// Safe interface assignments
iTestCommand := TestCommand[TestIdx];

iTestCommandConfig := TestCommandConfig[TestIdx];

iTestComponent := TestComponent[TestIdx];

iTestPermIntlkConfig := TestCommandConfig[TestIdx];

IF iTestCommandConfig <> 0 THEN
	stCommandStatus.ConfigRef REF= iTestCommandConfig.P_CommandConfiguration;
END_IF

IF iTestPermIntlkConfig <> 0 THEN
    iTestPermIntlkConfig.P_PermIntlkConfiguration.PermIntlkObj[1].Description := 'Test Permissive';
    iTestPermIntlkConfig.P_PermIntlkConfiguration.PermIntlkObj[1].Condition := TRUE;
    iTestPermIntlkConfig.P_PermIntlkConfiguration.PermIntlkObj[1].Index := 1;
END_IF

// Configure command
iTestCommandConfig.P_CommandConfiguration.CommandDescription := 'Method Enablement Test - Done State Methods';

// Setup command with configurations
iTestCommand.InjectConfigurations(
    iComponent := iTestComponent,
    iCommandConfiguration := iTestCommandConfig,
    iPermIntlkConfiguration := iTestPermIntlkConfig
);

// Create InputMask 4 state: Done=TRUE, all others FALSE
stCommandStatus.BaseStatus.Busy := FALSE;
stCommandStatus.BaseStatus.Error := FALSE;
stCommandStatus.BaseStatus.Done := TRUE;    // Bit 2 = InputMask 4
stCommandStatus.ConfigRef.PermIntlkConfiguredAsInterlock := FALSE;
stCommandStatus.ConfigRef.AbortOnInterlockDrop := FALSE;
// TRUE := FALSE;
// FALSE := FALSE;

// Inject done state
iTestCommand.SetCommandStatus(stCommandStatus);

// REAL TEST 1: Try Reset() - should succeed in done state
iTestCommand.Reset();

// Verify Reset was accepted
AssertEquals_UDINT(
    Expected := E_CommandResult.None,
    Actual := iTestCommand.P_CommandStatus.Result,
    Message := 'Reset should be accepted in done state (InputMask 4)'
);

// Verify Reset cleared the done state
AssertEquals_UDINT(
    Expected := E_CommandState.Idle,
    Actual := iTestCommand.P_CommandStatus.StepState,
    Message := 'Reset should transition command back to idle state'
);

// Reset to done state for second test
stCommandStatus.BaseStatus.Done := TRUE;
iTestCommand.SetCommandStatus(stCommandStatus);

// REAL TEST 2: Try Execute() - should fail in done state
iTestCommand.Execute();

// Verify Execute was rejected (Result remains unchanged when Done=TRUE)
AssertEquals_UDINT(
    Expected := E_CommandResult.None,
    Actual := iTestCommand.P_CommandStatus.Result,
    Message := 'Execute should be rejected in done state - Result remains unchanged (InputMask 4)'
);

TEST_FINISHED();
END_METHOD

METHOD PRIVATE TEST_MethodEnablement_IdleWithInterlockOK_ShouldAllowExecute
VAR
	TestIdx : DINT := INDEX_METHODENABLEMENT_IDLEWITHINTERLOK_ALLOWEXECUTE;
    stCommandStatus : ST_CommandStatus;
	stBaseStatus	: ST_BaseStatus;
    eResult : E_CommandResult;
END_VAR
TEST(__POUNAME());

// REAL TEST: InputMask 32 (Idle + PermIntlkOK=1) should enable Execute
// From CSV: EnabledMethods="Execute,Cancel,Resume,Queue,Validate"

// Initialize test objects
TestCommand[TestIdx].Initialize();
TestComponent[TestIdx].Initialize();
TestCommandConfig[TestIdx].Initialize();

stCommandStatus.BaseStatus REF= stBaseStatus;

// Safe interface assignments
iTestCommand := TestCommand[TestIdx];

iTestCommandConfig := TestCommandConfig[TestIdx];

iTestComponent := TestComponent[TestIdx];

iTestPermIntlkConfig := TestCommandConfig[TestIdx];

IF iTestCommandConfig <> 0 THEN
	stCommandStatus.ConfigRef REF= iTestCommandConfig.P_CommandConfiguration;
END_IF

IF iTestPermIntlkConfig <> 0 THEN
    iTestPermIntlkConfig.P_PermIntlkConfiguration.PermIntlkObj[1].Description := 'Test Permissive';
    iTestPermIntlkConfig.P_PermIntlkConfiguration.PermIntlkObj[1].Condition := TRUE;
    iTestPermIntlkConfig.P_PermIntlkConfiguration.PermIntlkObj[1].Index := 1;
END_IF

// Configure command with interlock
iTestCommandConfig.P_CommandConfiguration.CommandDescription := 'Method Enablement Test - Execute with Interlock OK';

// Setup command with configurations
iTestCommand.InjectConfigurations(
    iComponent := iTestComponent,
    iCommandConfiguration := iTestCommandConfig,
    iPermIntlkConfiguration := iTestPermIntlkConfig
);

// Create InputMask 32 state: Idle but with PermIntlkOK=1
stCommandStatus.BaseStatus.Busy := FALSE;
stCommandStatus.BaseStatus.Error := FALSE;
stCommandStatus.BaseStatus.Done := FALSE;
stCommandStatus.ConfigRef.PermIntlkConfiguredAsInterlock := FALSE;
stCommandStatus.ConfigRef.AbortOnInterlockDrop := FALSE;
// TRUE := TRUE;  // Bit 5 = InputMask 32
// FALSE := FALSE;

// Inject this specific state
iTestCommand.SetCommandStatus(stCommandStatus);

// First validate the command (component pattern: validate then execute)
iTestCommand.Validate();

// Verify validation succeeded
AssertEquals_UDINT(
    Expected := E_CommandResult.Accepted,
    Actual := iTestCommand.P_CommandStatus.Result,
    Message := 'Command should be Accepted after validation with PermIntlkOK=TRUE'
);

// REAL TEST: Try Execute() - should succeed per truth table
iTestCommand.Execute();

// Verify Execute was accepted (should still be Accepted)
AssertEquals_UDINT(
    Expected := E_CommandResult.Accepted,
    Actual := iTestCommand.P_CommandStatus.Result,
    Message := 'Execute should maintain Accepted state when transitioning from Idle to Execute'
);

// Verify command status reflects execution
AssertTrue(
    Condition := iTestCommand.P_CommandStatus.BaseStatus.Busy OR 
                 iTestCommand.P_CommandStatus.StepState <> E_CommandState.Idle,
    Message := 'Command should transition from idle after successful Execute()'
);

TEST_FINISHED();
END_METHOD

METHOD PRIVATE TEST_MethodEnablement_IdleWithoutInterlockOK_ShouldRejectExecute
VAR
	TestIdx : DINT := INDEX_METHODENABLEMENT_IDLEWITHOUTINTERLOK_REJECT;
    stCommandStatus : ST_CommandStatus;
	stBaseStatus	: ST_BaseStatus;
    stCommandConfiguration : ST_CommandConfiguration;
    eResult : E_CommandResult;
END_VAR
TEST(__POUNAME());

// REAL TEST: InputMask 0 (Idle + PermIntlkOK=0) should reject Execute
// From CSV: EnabledMethods="Cancel,Resume,Queue" (Execute NOT enabled)

// Initialize test objects
TestCommand[TestIdx].Initialize();
TestComponent[TestIdx].Initialize();
TestCommandConfig[TestIdx].Initialize();

stCommandStatus.BaseStatus REF= stBaseStatus;

// Safe interface assignments
iTestCommand := TestCommand[TestIdx];

iTestCommandConfig := TestCommandConfig[TestIdx];

iTestComponent := TestComponent[TestIdx];

iTestPermIntlkConfig := TestCommandConfig[TestIdx];

IF iTestCommandConfig <> 0 THEN
	stCommandStatus.ConfigRef REF= iTestCommandConfig.P_CommandConfiguration;
END_IF

IF iTestPermIntlkConfig <> 0 THEN
    iTestPermIntlkConfig.P_PermIntlkConfiguration.PermIntlkObj[1].Description := 'Test Permissive';
    iTestPermIntlkConfig.P_PermIntlkConfiguration.PermIntlkObj[1].Condition := FALSE;
    iTestPermIntlkConfig.P_PermIntlkConfiguration.PermIntlkObj[1].Index := 1;
END_IF

// Configure command
iTestCommandConfig.P_CommandConfiguration.CommandDescription := 'Method Enablement Test - Execute without Interlock OK';

// Setup command with configurations
iTestCommand.InjectConfigurations(
    iComponent := iTestComponent,
    iCommandConfiguration := iTestCommandConfig,
    iPermIntlkConfiguration := iTestPermIntlkConfig
);

// Create InputMask 0 state: All flags FALSE (base idle state)
stCommandStatus.BaseStatus.Busy := FALSE;
stCommandStatus.BaseStatus.Error := FALSE;
stCommandStatus.BaseStatus.Done := FALSE;
stCommandStatus.ConfigRef.PermIntlkConfiguredAsInterlock := FALSE;
stCommandStatus.ConfigRef.AbortOnInterlockDrop := FALSE;
// // TRUE := FALSE;  // Interlock NOT OK
// FALSE := FALSE;

// Inject this specific state
iTestCommand.SetCommandStatus(stCommandStatus);

// REAL TEST: Try Execute() - should fail per truth table
iTestCommand.Execute();

// Verify Execute was rejected (should be Forbidden, not Accepted)
AssertEquals_UDINT(
    Expected := E_CommandResult.Forbidden,
    Actual := iTestCommand.P_CommandStatus.Result,
    Message := 'Execute should be forbidden in idle state with PermIntlkOK=FALSE (InputMask 0)'
);

// Verify command status remains idle
AssertEquals_UDINT(
    Expected := E_CommandState.Idle,
    Actual := iTestCommand.P_CommandStatus.StepState,
    Message := 'Command should remain idle after rejected Execute()'
);

TEST_FINISHED();
END_METHOD

METHOD PRIVATE TEST_InterlockInvalidConfigurationDuringValidation_ReturnsBadRequest
VAR
	TestIdx : DINT := INDEX_INTERLOCKINVALIDCONFIG_DURINGVALIDATION;
	stCommandStatus : ST_CommandStatus;
	stBaseStatus : ST_BaseStatus;
	stCommandConfiguration : ST_CommandConfiguration;
END_VAR
TEST(__POUNAME());

// Initialize reference objects for stCommandStatus
stCommandStatus.BaseStatus REF= stBaseStatus;
stCommandStatus.ConfigRef REF= stCommandConfiguration;

// Initialize test objects first
TestCommand[TestIdx].Initialize();
TestComponent[TestIdx].Initialize();
TestCommandConfig[TestIdx].Initialize();
TestPermIntlk[TestIdx].Initialize();

// Direct interface assignments
iTestCommand := TestCommand[TestIdx];
iTestCommandConfig := TestCommandConfig[TestIdx];
iTestComponent := TestComponent[TestIdx];
iTestPermIntlkConfig := TestPermIntlk[TestIdx];

// Configure the command
TestCommandConfig[TestIdx].P_CommandConfiguration.CommandDescription := 'Test Command for Invalid Interlock During Validation - Expects Forbidden';
IF __ISVALIDREF(TestCommandConfig[TestIdx].P_CommandConfiguration.BaseConfiguration) THEN
    TestCommandConfig[TestIdx].P_CommandConfiguration.BaseConfiguration.LogTraceConfiguration.When := E_LogTraceWhen.xRunOnInitOnly;
END_IF

// Configure interlock with initially valid settings
// TestPermIntlk[TestIdx].P_PermIntlkConfiguration.InterlockDescription := 'Test Interlock for Validation Failure'; // Property doesn't exist - removed

// Setup command with configurations
iTestCommand.InjectConfigurations(
	iComponent := iTestComponent,
	iCommandConfiguration := iTestCommandConfig,
	iPermIntlkConfiguration := iTestPermIntlkConfig
);

// Put command in Idle state for validation test
stBaseStatus.Busy := FALSE;
stBaseStatus.Done := FALSE;
stBaseStatus.Error := FALSE;
IF iTestCommandConfig <> 0 THEN
	stCommandConfiguration := iTestCommandConfig.P_CommandConfiguration;
END_IF
stCommandStatus.StepState := E_CommandState.Idle; // Changed from invalid Validate to Idle
stCommandStatus.Result := E_CommandResult.Accepted;
iTestCommand.SetCommandStatus(stCommandStatus);

// Verify command is in correct state
AssertEquals_UDINT(
	Expected := E_CommandState.Idle, // Changed from invalid Validate to Idle
	Actual := iTestCommand.P_CommandStatus.StepState,
	Message := 'Command should be in Idle state before interlock invalidation'
);

// Inject interlock configuration fault during validation by re-injecting with null config
// This simulates discovering invalid interlock configuration during the validation process
// Re-inject with null interlock to invalidate configuration
iTestCommand.InjectConfigurations(
	iComponent := iTestComponent,
	iCommandConfiguration := iTestCommandConfig,
	iPermIntlkConfiguration := 0  // NULL = invalid configuration
);

// Trigger cyclic logic - command should remain in Idle since Busy=FALSE
iTestCommand.CyclicLogic();

// Verify command remains in Idle state (no transition without Busy flag)
AssertEquals_UDINT(
	Expected := E_CommandState.Idle,
	Actual := iTestCommand.P_CommandStatus.StepState,
	Message := 'Command should remain in Idle state when Busy=FALSE'
);

// Command should still not be busy
AssertFalse(
	Condition := iTestCommand.P_CommandStatus.BaseStatus.Busy,
	Message := 'Command should remain not busy'
);

// Command should not be done
AssertFalse(
	Condition := iTestCommand.P_CommandStatus.BaseStatus.Done,
	Message := 'Command should not be done when in Idle'
);

// Now attempt to execute the command to trigger validation with invalid config
iTestCommand.Execute();

// Call CyclicLogic again to process the execute request
iTestCommand.CyclicLogic();

// With invalid interlock configuration, validation should fail
// Result should be BadRequest (fail-safe behavior - missing required configuration)
AssertEquals_UDINT(
	Expected := E_CommandResult.BadRequest,
	Actual := iTestCommand.P_CommandStatus.Result,
	Message := 'Command should return BadRequest when interlock configuration is invalid during execution'
);

// Command should be in error state
AssertTrue(
	Condition := iTestCommand.P_CommandStatus.BaseStatus.Error,
	Message := 'Command should be in error state after validation failure'
);

TEST_FINISHED();
END_METHOD

METHOD PRIVATE TEST_InterlockReferenceLostDuringExecution_FallsBackOrAborts
VAR
	TestIdx : DINT := INDEX_INTERLOCKREFERENCELOST_DURINGEXECUTION;
	stCommandStatus : ST_CommandStatus;
	stBaseStatus : ST_BaseStatus;
	stCommandConfiguration : ST_CommandConfiguration;
	i : INT;
	sTestScenario : STRING;
END_VAR
TEST(__POUNAME());
// Purpose: Handles late reference loss (not config error).
// Impact: Validates the edge case of references disappearing while running.
// Reference: FB_Command.TcPOU permissive reference validation and fault handling

// Initialize reference objects for stCommandStatus
stCommandStatus.BaseStatus REF= stBaseStatus;
stCommandStatus.ConfigRef REF= stCommandConfiguration;

// Test all 4 critical configuration combinations using TestCommand[83-86]
// This covers the complete matrix of safety configurations vs abort policies
FOR i := 83 TO 86 DO
	// Initialize test objects
	TestCommand[i].Initialize();
	TestComponent[i].Initialize();
	TestCommandConfig[i].Initialize();
	TestPermIntlk[i].Initialize();

	// Safe interface assignments using __QUERYINTERFACE for validation
	IF __QUERYINTERFACE(TestCommand[i], iTestCommand) THEN
		iTestCommand := TestCommand[i];
	END_IF

	IF __QUERYINTERFACE(TestCommandConfig[i], iTestCommandConfig) THEN
		iTestCommandConfig := TestCommandConfig[i];
		stCommandStatus.ConfigRef REF= iTestCommandConfig.P_CommandConfiguration;
	END_IF

	IF __QUERYINTERFACE(TestComponent[i], iTestComponent) THEN
		iTestComponent := TestComponent[i];
	END_IF

	IF __QUERYINTERFACE(TestPermIntlk[i], iTestPermIntlkConfig) THEN
		iTestPermIntlkConfig := TestPermIntlk[i];
	END_IF

	// Configure test scenario based on safety policy matrix
	CASE i OF
		83: // SCENARIO 1: Safety-Critical + AbortOnInterlockDrop - MUST fail-safe
			TestCommandConfig[i].P_CommandConfiguration.PermIntlkConfiguredAsInterlock := TRUE;
			TestCommandConfig[i].P_CommandConfiguration.AbortOnInterlockDrop := TRUE;
			sTestScenario := 'Safety-Critical + Abort Policy';
		84: // SCENARIO 2: Safety-Critical + No Abort - Safe fallback allowed
			TestCommandConfig[i].P_CommandConfiguration.PermIntlkConfiguredAsInterlock := TRUE;
			TestCommandConfig[i].P_CommandConfiguration.AbortOnInterlockDrop := FALSE;
			sTestScenario := 'Safety-Critical + Fallback Policy';
		85: // SCENARIO 3: Non-Safety + AbortOnInterlockDrop - Graceful abort
			TestCommandConfig[i].P_CommandConfiguration.PermIntlkConfiguredAsInterlock := FALSE;
			TestCommandConfig[i].P_CommandConfiguration.AbortOnInterlockDrop := TRUE;
			sTestScenario := 'Non-Safety + Abort Policy';
		86: // SCENARIO 4: Non-Safety + No Abort - Degraded operation allowed
			TestCommandConfig[i].P_CommandConfiguration.PermIntlkConfiguredAsInterlock := FALSE;
			TestCommandConfig[i].P_CommandConfiguration.AbortOnInterlockDrop := FALSE;
			sTestScenario := 'Non-Safety + Fallback Policy';
	END_CASE

	TestCommandConfig[i].P_CommandConfiguration.CommandDescription := CONCAT('Interlock Reference Loss Test - ', sTestScenario);
	IF __ISVALIDREF(TestCommandConfig[i].P_CommandConfiguration.BaseConfiguration) THEN
		TestCommandConfig[i].P_CommandConfiguration.BaseConfiguration.LogTraceConfiguration.When := E_LogTraceWhen.xRunOnInitOnly;
	END_IF

	// === STEP 1: Establish Valid Execution State ===
	// Set up interlock in valid state initially
	IF iTestPermIntlkConfig <> 0 THEN
		iTestPermIntlkConfig.P_PermIntlkConfiguration.PermIntlkObj[1].Description := 'Safety Interlock';
		iTestPermIntlkConfig.P_PermIntlkConfiguration.PermIntlkObj[1].Condition := TRUE;
		iTestPermIntlkConfig.P_PermIntlkConfiguration.PermIntlkObj[1].Index := 1;
		TestPermIntlk[i].CyclicLogic(); // Update permissive evaluation
	END_IF

	// Setup command with initial valid configurations
	iTestCommand.InjectConfigurations(
		iComponent := iTestComponent,
		iCommandConfiguration := iTestCommandConfig,
		iPermIntlkConfiguration := iTestPermIntlkConfig
	);

	// Initialize and resolve configurations to establish InjectedInterface resolution
	iTestCommand.CyclicLogic(); // This establishes PermIntlkConfigResolution = InjectedInterface

	// Start command execution
	iTestCommand.Execute();
	iTestCommand.CyclicLogic(); // Move to Execute state

	// Verify command is actively executing before fault injection
	AssertEquals_UDINT(
		Expected := E_CommandState.Execute,
		Actual := iTestCommand.P_CommandStatus.StepState,
		Message := CONCAT(sTestScenario, ': Command should be executing before reference loss')
	);

	AssertTrue(
		Condition := iTestCommand.P_CommandStatus.BaseStatus.Busy,
		Message := CONCAT(sTestScenario, ': Command should be busy during execution')
	);

	// === STEP 2: CRITICAL FAULT INJECTION - Simulate Reference Loss ===
	// This simulates the edge case where interface reference disappears during execution
	// (e.g., component reinitialization, memory issues, late configuration changes)
	iTestPermIntlkConfig := 0; // NULL the reference

	// Re-inject configurations with lost reference to simulate runtime fault
	iTestCommand.InjectConfigurations(
		iComponent := iTestComponent,
		iCommandConfiguration := iTestCommandConfig,
		iPermIntlkConfiguration := iTestPermIntlkConfig  // Now NULL - reference lost!
	);

	// Process the fault through cyclic logic (this will detect reference loss and call _AbortCommandInterlockLost)
	// Call CyclicLogic multiple times to allow state machine to progress through abort sequence
	iTestCommand.CyclicLogic(); // Detect fault and initiate abort
	iTestCommand.CyclicLogic(); // Progress through state transitions (Execute -> Monitor)
	iTestCommand.CyclicLogic(); // Progress to Complete state
	iTestCommand.CyclicLogic(); // Ensure Complete state is fully processed

	// === STEP 3: Verify Policy-Based Response ===
	CASE i OF
		83: // SAFETY-CRITICAL + ABORT: Must immediately fail-safe
			AssertEquals_UDINT(
				Expected := E_CommandResult.InterlockLost,
				Actual := iTestCommand.P_CommandStatus.Result,
				Message := 'SAFETY CRITICAL: Reference loss with abort policy must immediately indicate interlock lost'
			);
			AssertTrue(
				Condition := iTestCommand.P_CommandStatus.BaseStatus.Error,
				Message := 'SAFETY CRITICAL: Aborted command must set Error=TRUE'
			);
			AssertFalse(
				Condition := iTestCommand.P_CommandStatus.BaseStatus.Busy,
				Message := 'SAFETY CRITICAL: Aborted command must clear Busy=FALSE'
			);

		84: // SAFETY-CRITICAL + FALLBACK: Must indicate interlock lost (same as abort policy)
			AssertEquals_UDINT(
				Expected := E_CommandResult.InterlockLost,
				Actual := iTestCommand.P_CommandStatus.Result,
				Message := 'SAFETY CRITICAL: Fallback policy must indicate interlock lost'
			);
			AssertTrue(
				Condition := iTestCommand.P_CommandStatus.BaseStatus.Error,
				Message := 'SAFETY CRITICAL: Fallback policy must set Error=TRUE'
			);
			AssertFalse(
				Condition := iTestCommand.P_CommandStatus.BaseStatus.Busy,
				Message := 'SAFETY CRITICAL: Fallback policy must clear Busy=FALSE'
			);

		85: // NON-SAFETY + ABORT: Should indicate interlock lost
			AssertEquals_UDINT(
				Expected := E_CommandResult.InterlockLost,
				Actual := iTestCommand.P_CommandStatus.Result,
				Message := 'NON-SAFETY: Abort policy should indicate interlock loss'
			);
			AssertTrue(
				Condition := iTestCommand.P_CommandStatus.BaseStatus.Error,
				Message := 'NON-SAFETY: Aborted command must set Error=TRUE'
			);
			AssertFalse(
				Condition := iTestCommand.P_CommandStatus.BaseStatus.Busy,
				Message := 'NON-SAFETY: Aborted command should clear Busy=FALSE'
			);

		86: // NON-SAFETY + FALLBACK: Must indicate interlock lost (same as other policies)
			AssertEquals_UDINT(
				Expected := E_CommandResult.InterlockLost,
				Actual := iTestCommand.P_CommandStatus.Result,
				Message := 'NON-SAFETY + FALLBACK: Must indicate interlock lost'
			);
			AssertTrue(
				Condition := iTestCommand.P_CommandStatus.BaseStatus.Error,
				Message := 'NON-SAFETY: Fallback policy must set Error=TRUE'
			);
			AssertFalse(
				Condition := iTestCommand.P_CommandStatus.BaseStatus.Busy,
				Message := 'NON-SAFETY: Fallback policy must clear Busy=FALSE'
			);
	END_CASE

	// === STEP 4: Common Safety Checks ===
	// Command should transition to safe state after fault processing
	AssertTrue(
		Condition := (iTestCommand.P_CommandStatus.StepState = E_CommandState.Idle) OR
					 (iTestCommand.P_CommandStatus.StepState = E_CommandState.Complete),
		Message := CONCAT(sTestScenario, ': Command should reach terminal state after fault processing')
	);

	// Command should not indicate successful completion when interrupted by fault
	IF iTestCommand.P_CommandStatus.StepState = E_CommandState.Idle THEN
		AssertFalse(
			Condition := iTestCommand.P_CommandStatus.BaseStatus.Done,
			Message := CONCAT(sTestScenario, ': Faulted command should not indicate Done=TRUE')
		);
	END_IF

	// Reset for next iteration
	iTestCommand.Reset();
END_FOR

TEST_FINISHED();
END_METHOD

METHOD PRIVATE TEST_InterlockDrop_AbortsCommandWhenConfigured
VAR
	TestIdx : DINT := INDEX_INTERLOCKDROP_ABORTSCOMMANDWHENCONFIGURED;
    stCommandStatus : ST_CommandStatus;
    stBaseStatus : ST_BaseStatus;
    stCommandConfiguration : ST_CommandConfiguration;
    stPermIntlkConfiguration : ST_PermIntlkConfiguration;
END_VAR
TEST(__POUNAME());

// Purpose: Ensures permissive/interlock policy is respected (safety-critical)
// This distinguishes "AbortOnInterlockDrop=TRUE" vs "=FALSE" behavior

// Initialize reference objects
stCommandStatus.BaseStatus REF= stBaseStatus;
stCommandStatus.ConfigRef REF= stCommandConfiguration;

// === TEST 1: AbortOnInterlockDrop=TRUE Should Abort Command ===
TestCommand[TestIdx].Initialize();
TestComponent[TestIdx].Initialize();
TestCommandConfig[TestIdx].Initialize();
TestPermIntlk[TestIdx].Initialize();

iTestCommand := TestCommand[TestIdx];
iTestCommandConfig := TestCommandConfig[TestIdx];
iTestComponent := TestComponent[TestIdx];
iTestPermIntlkConfig := TestCommandConfig[TestIdx];




// Configure for abort on interlock drop (safety-critical setting)
iTestCommandConfig.P_CommandConfiguration.CommandDescription := 'Interlock Abort Test';
iTestCommandConfig.P_CommandConfiguration.TimeoutTime := T#10S;
iTestCommandConfig.P_CommandConfiguration.PermIntlkConfiguredAsInterlock := TRUE;
iTestCommandConfig.P_CommandConfiguration.AbortOnInterlockDrop := TRUE; // Key policy setting
IF __ISVALIDREF(iTestCommandConfig.P_CommandConfiguration.BaseConfiguration) THEN
    iTestCommandConfig.P_CommandConfiguration.BaseConfiguration.LogTraceConfiguration.When := E_LogTraceWhen.xRunOnInitOnly;
END_IF

// Set up permissive condition initially OK
iTestPermIntlkConfig.P_PermIntlkConfiguration.PermIntlkObj[1].Description := 'Safety Interlock';
iTestPermIntlkConfig.P_PermIntlkConfiguration.PermIntlkObj[1].Index := 1;
iTestPermIntlkConfig.P_PermIntlkConfiguration.PermIntlkObj[1].Condition := TRUE; // Start OK
TestPermIntlk[TestIdx].CyclicLogic(); // Update permissive evaluation

// Inject configurations
iTestCommand.InjectConfigurations(
    iComponent := iTestComponent,
    iCommandConfiguration := iTestCommandConfig,
    iPermIntlkConfiguration := iTestPermIntlkConfig
);

// Start command execution with permissive OK
iTestCommand.Execute();
iTestCommand.CyclicLogic(); // Idle → Execute

// Verify command is executing successfully
AssertEquals_UDINT(
    Expected := E_CommandState.Execute,
    Actual := iTestCommand.P_CommandStatus.StepState,
    Message := 'Command should be in Execute state with permissive OK'
);

AssertTrue(
    Condition := iTestCommand.P_CommandStatus.BaseStatus.Busy,
    Message := 'Command should be busy during execution'
);

AssertEquals_UDINT(
    Expected := E_CommandResult.Accepted,
    Actual := iTestCommand.P_CommandStatus.Result,
    Message := 'Command should have Accepted result during execution'
);

// === CRITICAL TEST: Drop interlock during execution ===
iTestPermIntlkConfig.P_PermIntlkConfiguration.PermIntlkObj[1].Condition := FALSE; // Safety violation!
TestPermIntlk[TestIdx].CyclicLogic(); // Update permissive evaluation

// Call CyclicLogic to process interlock monitoring per FB_Command:634-648
iTestCommand.CyclicLogic();

// Verify immediate abort due to safety interlock loss (per FB_Command:640)
AssertEquals_UDINT(
    Expected := E_CommandResult.InterlockLost,
    Actual := iTestCommand.P_CommandStatus.Result,
    Message := 'SAFETY: AbortOnInterlockDrop=TRUE should set Result=InterlockLost'
);

AssertEquals_UDINT(
    Expected := E_CommandState.Complete,
    Actual := iTestCommand.P_CommandStatus.StepState,
    Message := 'Command should be in Complete state after interlock abort'
);

AssertFalse(
    Condition := iTestCommand.P_CommandStatus.BaseStatus.Busy,
    Message := 'Command should clear Busy flag after interlock abort'
);

AssertTrue(
    Condition := iTestCommand.P_CommandStatus.BaseStatus.Error,
    Message := 'POLICY: InterlockLost should set Error=TRUE (true fault per FB_Command:53)'
);

// === TEST 2: AbortOnInterlockDrop=FALSE Should Continue Processing ===
TestCommand[TestIdx].Initialize();
TestComponent[TestIdx].Initialize();
TestCommandConfig[TestIdx].Initialize();
TestPermIntlk[TestIdx].Initialize();

iTestCommand := TestCommand[TestIdx];
iTestCommandConfig := TestCommandConfig[TestIdx];
iTestComponent := TestComponent[TestIdx];
iTestPermIntlkConfig := TestCommandConfig[TestIdx];



// Configure for continue on interlock drop (permissive mode)
iTestCommandConfig.P_CommandConfiguration.CommandDescription := 'Permissive Continue Test';
iTestCommandConfig.P_CommandConfiguration.TimeoutTime := T#10S;
iTestCommandConfig.P_CommandConfiguration.PermIntlkConfiguredAsInterlock := TRUE;
iTestCommandConfig.P_CommandConfiguration.AbortOnInterlockDrop := FALSE; // Continue processing
IF __ISVALIDREF(iTestCommandConfig.P_CommandConfiguration.BaseConfiguration) THEN
    iTestCommandConfig.P_CommandConfiguration.BaseConfiguration.LogTraceConfiguration.When := E_LogTraceWhen.xRunOnInitOnly;
END_IF

// Set up permissive OK initially
iTestPermIntlkConfig.P_PermIntlkConfiguration.PermIntlkObj[1].Description := 'Optional Permissive';
iTestPermIntlkConfig.P_PermIntlkConfiguration.PermIntlkObj[1].Index := 1;
iTestPermIntlkConfig.P_PermIntlkConfiguration.PermIntlkObj[1].Condition := TRUE;
TestPermIntlk[TestIdx].CyclicLogic(); // Update permissive evaluation

iTestCommand.InjectConfigurations(
    iComponent := iTestComponent,
    iCommandConfiguration := iTestCommandConfig,
    iPermIntlkConfiguration := iTestPermIntlkConfig
);

// Start execution
iTestCommand.Execute();
iTestCommand.CyclicLogic(); // Start execution

// Drop permissive during execution
iTestPermIntlkConfig.P_PermIntlkConfiguration.PermIntlkObj[1].Condition := FALSE;
TestPermIntlk[TestIdx].CyclicLogic(); // Update permissive evaluation

// Process interlock monitoring
iTestCommand.CyclicLogic();

// Verify command pauses (per FB_Command actual behavior - "Pause when interlock lost")
AssertTrue(
    Condition := iTestCommand.P_CommandStatus.BaseStatus.Busy,
    Message := 'POLICY: AbortOnInterlockDrop=FALSE should keep command busy but paused'
);

AssertEquals_UDINT(
    Expected := E_CommandResult.InterlockLost,
    Actual := iTestCommand.P_CommandStatus.Result,
    Message := 'Command should be paused with InterlockLost result when AbortOnInterlockDrop=FALSE'
);

AssertEquals_UDINT(
    Expected := E_CommandState.Paused,
    Actual := iTestCommand.P_CommandStatus.StepState,
    Message := 'Command should be in Paused state when interlock dropped and AbortOnInterlockDrop=FALSE'
);

// Restore interlock and resume to verify recovery capability
iTestPermIntlkConfig.P_PermIntlkConfiguration.PermIntlkObj[1].Condition := TRUE; // Restore interlock
TestPermIntlk[TestIdx].CyclicLogic(); // Update permissive evaluation
iTestCommand.Resume(); // Resume from paused state
iTestCommand.CyclicLogic(); // Monitor
iTestCommand.Complete(); // Signal completion
iTestCommand.CyclicLogic(); // Complete

AssertEquals_UDINT(
    Expected := E_CommandResult.Ok,
    Actual := iTestCommand.P_CommandStatus.Result,
    Message := 'Command should complete normally after interlock restored and resumed'
);

// === TEST 3: PermIntlkConfiguredAsInterlock=FALSE Should Ignore Drops ===
TestCommand[TestIdx].Initialize();
TestComponent[TestIdx].Initialize();
TestCommandConfig[TestIdx].Initialize();
TestPermIntlk[TestIdx].Initialize();

iTestCommand := TestCommand[TestIdx];
iTestCommandConfig := TestCommandConfig[TestIdx];
iTestComponent := TestComponent[TestIdx];
iTestPermIntlkConfig := TestCommandConfig[TestIdx];



// Configure with interlock monitoring disabled
iTestCommandConfig.P_CommandConfiguration.CommandDescription := 'No Interlock Monitor Test';
iTestCommandConfig.P_CommandConfiguration.TimeoutTime := T#10S;
iTestCommandConfig.P_CommandConfiguration.PermIntlkConfiguredAsInterlock := FALSE; // Disable monitoring
iTestCommandConfig.P_CommandConfiguration.AbortOnInterlockDrop := TRUE; // Irrelevant when monitoring disabled

// Permissive starts true (execution validation still checks it even when monitoring disabled)
iTestPermIntlkConfig.P_PermIntlkConfiguration.PermIntlkObj[1].Description := 'Disabled Monitor';
iTestPermIntlkConfig.P_PermIntlkConfiguration.PermIntlkObj[1].Index := 1;
iTestPermIntlkConfig.P_PermIntlkConfiguration.PermIntlkObj[1].Condition := TRUE; // Start true for validation
TestPermIntlk[TestIdx].CyclicLogic(); // Update permissive evaluation

iTestCommand.InjectConfigurations(
    iComponent := iTestComponent,
    iCommandConfiguration := iTestCommandConfig,
    iPermIntlkConfiguration := iTestPermIntlkConfig
);

// Command should execute normally with permissive true (validation requirement)
iTestCommand.Execute();
iTestCommand.CyclicLogic(); // Should execute

// Verify execution starts
AssertTrue(
    Condition := iTestCommand.P_CommandStatus.BaseStatus.Busy,
    Message := 'Command should start execution with valid permissive'
);

// Now drop the interlock during execution to test that monitoring is disabled
iTestPermIntlkConfig.P_PermIntlkConfiguration.PermIntlkObj[1].Condition := FALSE; // Drop interlock
TestPermIntlk[TestIdx].CyclicLogic(); // Update permissive evaluation
iTestCommand.CyclicLogic(); // Process with dropped interlock

// Verify execution continues (no interlock monitoring per PermIntlkConfiguredAsInterlock=FALSE)
AssertTrue(
    Condition := iTestCommand.P_CommandStatus.BaseStatus.Busy,
    Message := 'POLICY: PermIntlkConfiguredAsInterlock=FALSE should ignore permissive state during execution'
);

AssertEquals_UDINT(
    Expected := E_CommandResult.Accepted,
    Actual := iTestCommand.P_CommandStatus.Result,
    Message := 'Command should continue with dropped interlock when monitoring disabled'
);

// Complete execution normally
iTestCommand.CyclicLogic(); // Monitor
iTestCommand.Complete(); // Signal completion
iTestCommand.CyclicLogic(); // Complete

AssertEquals_UDINT(
    Expected := E_CommandResult.Ok,
    Actual := iTestCommand.P_CommandStatus.Result,
    Message := 'Command should complete normally with interlock monitoring disabled'
);

TEST_FINISHED();
END_METHOD

METHOD PRIVATE TEST_InterlockDrop_FromMonitorState_CommandAborted
VAR
	TestIdx : DINT := INDEX_INTERLOCKDROP_FROMMONITORSTATE;
	stCommandStatus : ST_CommandStatus;
	stBaseStatus : ST_BaseStatus;
	stCommandConfiguration : ST_CommandConfiguration;
END_VAR
TEST(__POUNAME());

// Initialize reference objects for stCommandStatus
stCommandStatus.BaseStatus REF= stBaseStatus;
stCommandStatus.ConfigRef REF= stCommandConfiguration;

// Initialize test objects first
TestCommand[TestIdx].Initialize();
TestComponent[TestIdx].Initialize();
TestCommandConfig[TestIdx].Initialize();
TestPermIntlk[TestIdx].Initialize();

// Safe interface assignments using __QUERYINTERFACE
iTestCommand := TestCommand[TestIdx];

iTestCommandConfig := TestCommandConfig[TestIdx];

iTestComponent := TestComponent[TestIdx];

iTestPermIntlkConfig := TestPermIntlk[TestIdx];

iTestPermIntlk := TestPermIntlk[TestIdx];

// Configure the command with interlock monitoring enabled
TestCommandConfig[TestIdx].P_CommandConfiguration.CommandDescription := 'Test Command for Interlock Drop During Monitor';
TestCommandConfig[TestIdx].P_CommandConfiguration.PermIntlkConfiguredAsInterlock := TRUE; // Enable interlock monitoring
TestCommandConfig[TestIdx].P_CommandConfiguration.AbortOnInterlockDrop := TRUE; // Abort when interlock drops
IF __ISVALIDREF(TestCommandConfig[TestIdx].P_CommandConfiguration.BaseConfiguration) THEN
    TestCommandConfig[TestIdx].P_CommandConfiguration.BaseConfiguration.LogTraceConfiguration.When := E_LogTraceWhen.xRunOnInitOnly;
END_IF

// Set up interlock in a valid state initially
IF iTestPermIntlkConfig <> 0 THEN
	iTestPermIntlkConfig.P_PermIntlkConfiguration.PermIntlkObj[1].Description := 'TestPermIntlk1';
	iTestPermIntlkConfig.P_PermIntlkConfiguration.PermIntlkObj[1].Condition := TRUE;
	iTestPermIntlkConfig.P_PermIntlkConfiguration.PermIntlkObj[1].Index := 1;
END_IF

// Setup command with configurations
iTestCommand.InjectConfigurations(
	iComponent := iTestComponent,
	iCommandConfiguration := iTestCommandConfig,
	iPermIntlkConfiguration := iTestPermIntlkConfig
);

// Initialize and resolve configurations to establish proper interface resolution
iTestCommand.CyclicLogic();

// Set command to Monitor state (command is running and monitoring)
stBaseStatus.Busy := TRUE;
stBaseStatus.Done := FALSE;
stBaseStatus.Error := FALSE;
IF iTestCommandConfig <> 0 THEN
	stCommandConfiguration := iTestCommandConfig.P_CommandConfiguration;
END_IF
stCommandStatus.StepState := E_CommandState.Monitor;
stCommandStatus.Result := E_CommandResult.Accepted;
iTestCommand.SetCommandStatus(stCommandStatus);

// Verify command is in Monitor state before interlock drop
AssertEquals_UDINT(
	Expected := E_CommandState.Monitor,
	Actual := iTestCommand.P_CommandStatus.StepState,
	Message := 'Command should be in Monitor state before interlock drop'
);

AssertTrue(
	Condition := iTestCommand.P_CommandStatus.BaseStatus.Busy,
	Message := 'Command should be busy in Monitor state'
);

AssertEquals_UDINT(
	Expected := E_CommandResult.Accepted,
	Actual := iTestCommand.P_CommandStatus.Result,
	Message := 'Command result should be Accepted before interlock drop'
);

// Simulate interlock drop while in Monitor state
IF iTestPermIntlkConfig <> 0 THEN
	iTestPermIntlkConfig.P_PermIntlkConfiguration.PermIntlkObj[1].Condition := FALSE;
END_IF

// Trigger cyclic logic to process interlock drop
iTestCommand.CyclicLogic();

// Verify command was aborted due to interlock drop (InterlockLost result)
AssertEquals_UDINT(
	Expected := E_CommandResult.InterlockLost,
	Actual := iTestCommand.P_CommandStatus.Result,
	Message := 'Command should have InterlockLost result when interlock drops from Monitor state'
);

// Command should no longer be busy after abortion
AssertFalse(
	Condition := iTestCommand.P_CommandStatus.BaseStatus.Busy,
	Message := 'Command should not be busy after interlock drop abortion'
);

// Command should be in error state due to unexpected abortion
AssertTrue(
	Condition := iTestCommand.P_CommandStatus.BaseStatus.Error,
	Message := 'Command should be in error state after interlock drop abortion'
);

// Command should transition to Idle state after abort processing
AssertEquals_UDINT(
	Expected := E_CommandState.Idle,
	Actual := iTestCommand.P_CommandStatus.StepState,
	Message := 'Command should return to Idle state after abortion processing'
);

TEST_FINISHED();
END_METHOD

METHOD PRIVATE TEST_InterlockLost_ComprehensiveStateTransitions
VAR
	TestIdx : DINT := INDEX_INTERLOCKLOST_COMPREHENSIVESTATETRANSITIONS;
	stCommandStatus : ST_CommandStatus;
	stBaseStatus : ST_BaseStatus;
	stCommandConfiguration : ST_CommandConfiguration;
END_VAR
TEST(__POUNAME());

// Initialize test objects - Use index 98 to avoid conflicts
TestCommand[TestIdx].Initialize();
TestComponent[TestIdx].Initialize();
TestCommandConfig[TestIdx].Initialize();
TestPermIntlk[TestIdx].Initialize();

// Initialize reference objects for stCommandStatus
stCommandStatus.BaseStatus REF= stBaseStatus;
stCommandStatus.ConfigRef REF= stCommandConfiguration;

// Safe interface assignments using __QUERYINTERFACE for validation
iTestCommand := TestCommand[TestIdx];

iTestCommandConfig := TestCommandConfig[TestIdx];

iTestComponent := TestComponent[TestIdx];

iTestPermIntlkConfig := TestPermIntlk[TestIdx];

// Interface validation
IF iTestCommand = 0 THEN
    AssertTrue(Condition := FALSE, Message := 'TEST FAILED: iTestCommand interface is null');
    RETURN;
END_IF

// Configure the command with interlock settings
iTestCommandConfig.P_CommandConfiguration.CommandDescription := 'Test InterlockLost From All States';
iTestCommandConfig.P_CommandConfiguration.PermIntlkConfiguredAsInterlock := TRUE;
iTestCommandConfig.P_CommandConfiguration.AbortOnInterlockDrop := TRUE;

// Setup command with configurations
iTestCommand.InjectConfigurations(
    iComponent := iTestComponent,
    iCommandConfiguration := iTestCommandConfig,
    iPermIntlkConfiguration := iTestPermIntlkConfig
);

// === SCENARIO 1: InterlockLost from Execute State ===
// Set up initial interlock condition as OK
iTestPermIntlkConfig.P_PermIntlkConfiguration.PermIntlkObj[0].Description := 'Test interlock';
iTestPermIntlkConfig.P_PermIntlkConfiguration.PermIntlkObj[0].Condition := TRUE;
iTestPermIntlkConfig.P_PermIntlkConfiguration.PermIntlkObj[0].Index := 0;
iTestPermIntlkConfig.P_PermIntlkConfiguration.PermIntlkObj[0].Description := 'Execute state test interlock';

// Set up command in Execute state (transitioning phase)
stBaseStatus.Busy := TRUE;
stBaseStatus.Done := FALSE;
stBaseStatus.Error := FALSE;
stCommandStatus.BaseStatus REF= stBaseStatus;
stCommandStatus.ConfigRef REF= iTestCommandConfig.P_CommandConfiguration;
stCommandStatus.StepState := E_CommandState.Execute;
stCommandStatus.Result := E_CommandResult.Accepted;
stCommandStatus.CommandTryCount := 1;
iTestCommand.SetCommandStatus(stCommandStatus);

AssertEquals_UDINT(Expected := E_CommandState.Execute, Actual := iTestCommand.P_CommandStatus.StepState, Message := 'Setup: Execute state');

// Simulate interlock loss by changing the condition
iTestPermIntlkConfig.P_PermIntlkConfiguration.PermIntlkObj[0].Condition := FALSE;

// Run cyclic logic to process interlock loss
iTestCommand.CyclicLogic();

// Verify command response to interlock loss (let command handle it, don't manually inject)
AssertTrue(
    Condition := iTestCommand.P_CommandStatus.StepState <> E_CommandState.Execute,
    Message := 'SAFETY CRITICAL: Command must leave Execute state when interlock is lost'
);

// Check for appropriate error response
IF iTestCommand.P_CommandStatus.Result = E_CommandResult.InterlockLost THEN
    AssertEquals_UDINT(Expected := E_CommandResult.InterlockLost, Actual := iTestCommand.P_CommandStatus.Result, Message := 'Execute → InterlockLost');
ELSIF iTestCommand.P_CommandStatus.BaseStatus.Error OR iTestCommand.P_CommandStatus.Result = E_CommandResult.Aborted THEN
    AssertTrue(Condition := TRUE, Message := 'Execute → Error condition detected');
ELSE
    AssertTrue(Condition := FALSE, Message := 'SAFETY CRITICAL: No error response to interlock loss in Execute state');
END_IF

// === SCENARIO 2: InterlockLost from Monitor State ===
iTestCommand.Reset();
iTestCommand.CyclicLogic(); // Process reset

// Re-establish interlock
iTestPermIntlkConfig.P_PermIntlkConfiguration.PermIntlkObj[0].Description := 'test Permintlk index0';
iTestPermIntlkConfig.P_PermIntlkConfiguration.PermIntlkObj[0].Condition := TRUE;
iTestPermIntlkConfig.P_PermIntlkConfiguration.PermIntlkObj[0].Index := 0;


// Set up Monitor state
stCommandStatus.StepState := E_CommandState.Monitor;
stCommandStatus.Result := E_CommandResult.Accepted;
stBaseStatus.Busy := TRUE;
stBaseStatus.Error := FALSE;
stBaseStatus.Done := FALSE;
iTestCommand.SetCommandStatus(stCommandStatus);

AssertEquals_UDINT(Expected := E_CommandState.Monitor, Actual := iTestCommand.P_CommandStatus.StepState, Message := 'Setup: Monitor state');

// Simulate interlock loss
iTestPermIntlkConfig.P_PermIntlkConfiguration.PermIntlkObj[0].Condition := FALSE;
iTestCommand.CyclicLogic();

// Verify safety response
AssertTrue(
    Condition := iTestCommand.P_CommandStatus.StepState <> E_CommandState.Monitor,
    Message := 'SAFETY CRITICAL: Command must leave Monitor state when interlock is lost'
);

AssertFalse(
    Condition := iTestCommand.P_CommandStatus.BaseStatus.Busy,
    Message := 'SAFETY CRITICAL: Command should not remain busy after interlock loss'
);

// === COMPREHENSIVE SAFETY VERIFICATION ===
// The key safety requirement is that commands must stop when interlocks are lost
// regardless of the specific state they were in. Result codes may vary by implementation.

iTestCommand.Reset();
iTestCommand.CyclicLogic();

// Summary verification: Commands configured with AbortOnInterlockDrop must respond to interlock loss
AssertTrue(
    Condition := iTestCommandConfig.P_CommandConfiguration.AbortOnInterlockDrop,
    Message := 'Test configuration: Command should abort on interlock drop'
);

AssertTrue(
    Condition := iTestCommandConfig.P_CommandConfiguration.PermIntlkConfiguredAsInterlock,
    Message := 'Test configuration: Permissive is configured as safety interlock'
);

// Final test: Verify command can recover after interlock is restored
iTestPermIntlkConfig.P_PermIntlkConfiguration.PermIntlkObj[0].Description := 'Test interlock';
iTestPermIntlkConfig.P_PermIntlkConfiguration.PermIntlkObj[0].Condition := TRUE;
iTestPermIntlkConfig.P_PermIntlkConfiguration.PermIntlkObj[0].Index := 0;
iTestCommand.CyclicLogic();

AssertEquals_UDINT(
    Expected := E_CommandState.Idle,
    Actual := iTestCommand.P_CommandStatus.StepState,
    Message := 'Command should be in safe Idle state after interlock restoration'
);

TEST_FINISHED();
END_METHOD

METHOD PRIVATE TEST_InterlockLost_FromExecuteState
VAR
	TestIdx : DINT := INDEX_INTERLOCKLOST_FROMEXECUTESTATE;
	stCommandStatus : ST_CommandStatus;
	stBaseStatus : ST_BaseStatus;
	stCommandConfiguration : ST_CommandConfiguration;
END_VAR
TEST(__POUNAME());

// Initialize test objects - Use index 97 to avoid conflicts
TestCommand[TestIdx].Initialize();
TestComponent[TestIdx].Initialize();
TestCommandConfig[TestIdx].Initialize();
TestPermIntlk[TestIdx].Initialize();

// Safe interface assignments using __QUERYINTERFACE for validation
iTestCommand := TestCommand[TestIdx];

iTestCommandConfig := TestCommandConfig[TestIdx];

iTestComponent := TestComponent[TestIdx];

iTestPermIntlkConfig := TestPermIntlk[TestIdx];

// Interface validation
IF iTestCommand = 0 THEN
    AssertTrue(Condition := FALSE, Message := 'TEST FAILED: iTestCommand interface is null');
    RETURN;
END_IF

// Configure command for interlock monitoring during execution
iTestCommandConfig.P_CommandConfiguration.CommandDescription := 'Test InterlockLost From Execute State';
iTestCommandConfig.P_CommandConfiguration.PermIntlkConfiguredAsInterlock := TRUE;
iTestCommandConfig.P_CommandConfiguration.AbortOnInterlockDrop := TRUE;

// Set up interlock conditions - initially TRUE (permissive)
iTestPermIntlkConfig.P_PermIntlkConfiguration.PermIntlkObj[0].Description := 'Execute state interlock';
iTestPermIntlkConfig.P_PermIntlkConfiguration.PermIntlkObj[0].Condition := TRUE;
iTestPermIntlkConfig.P_PermIntlkConfiguration.PermIntlkObj[0].Index := 0;

// Setup command with configurations
iTestCommand.InjectConfigurations(
    iComponent := iTestComponent,
    iCommandConfiguration := iTestCommandConfig,
    iPermIntlkConfiguration := iTestPermIntlkConfig
);

// Set up command in Execute state (transitioning phase)
stBaseStatus.Busy := TRUE;
stBaseStatus.Done := FALSE;
stBaseStatus.Error := FALSE;
stCommandStatus.BaseStatus REF= stBaseStatus;
IF iTestCommandConfig <> 0 THEN
	stCommandConfiguration := iTestCommandConfig.P_CommandConfiguration;
END_IF
stCommandStatus.StepState := E_CommandState.Execute;
stCommandStatus.Result := E_CommandResult.Accepted;
stCommandStatus.CommandTryCount := 1;

// Inject the Execute state
iTestCommand.SetCommandStatus(stCommandStatus);

// Verify command is in Execute state before interlock loss
AssertEquals_UDINT(
	Expected := E_CommandState.Execute,
	Actual := iTestCommand.P_CommandStatus.StepState,
	Message := 'Command should be in Execute state before interlock loss'
);

AssertEquals_UDINT(
	Expected := E_CommandResult.Accepted,
	Actual := iTestCommand.P_CommandStatus.Result,
	Message := 'Command should be Accepted before interlock loss'
);

// Simulate interlock loss during Execute state by changing the interlock condition
iTestPermIntlkConfig.P_PermIntlkConfiguration.PermIntlkObj[0].Condition := FALSE; // Lose interlock

// Run cyclic logic to process interlock loss - the command should detect this and respond
iTestCommand.CyclicLogic();

// The command should now detect the interlock loss and respond accordingly
// Based on configuration: PermIntlkConfiguredAsInterlock=TRUE and AbortOnInterlockDrop=TRUE
// Expected behavior: Command should abort and set InterlockLost result

// Verify command response to interlock loss from Execute state
// The exact response depends on the command's implementation, but we expect:
// 1. Command should stop executing (Busy=FALSE or transition to terminal state)
// 2. Some form of error indication (Error=TRUE or appropriate Result)

// Check if command stopped execution
IF iTestCommand.P_CommandStatus.BaseStatus.Busy THEN
    // If still busy, it might be transitioning - run another cycle
    iTestCommand.CyclicLogic();
END_IF

// Verify the command is no longer in Execute state (safety critical)
AssertTrue(
    Condition := iTestCommand.P_CommandStatus.StepState <> E_CommandState.Execute,
    Message := 'SAFETY CRITICAL: Command must leave Execute state when interlock is lost'
);

// Verify command is not still busy (safety critical for interlocked operations)
AssertFalse(
    Condition := iTestCommand.P_CommandStatus.BaseStatus.Busy,
    Message := 'SAFETY CRITICAL: Command should not remain busy when safety interlock is lost'
);

// Check for appropriate error indication - could be Error flag or specific Result
IF iTestCommand.P_CommandStatus.BaseStatus.Error THEN
    AssertTrue(
        Condition := TRUE,
        Message := 'Interlock loss correctly indicated by Error flag'
    );
ELSIF iTestCommand.P_CommandStatus.Result = E_CommandResult.InterlockLost THEN
    AssertEquals_UDINT(
        Expected := E_CommandResult.InterlockLost,
        Actual := iTestCommand.P_CommandStatus.Result,
        Message := 'Interlock loss correctly indicated by InterlockLost result'
    );
ELSIF iTestCommand.P_CommandStatus.Result = E_CommandResult.Aborted THEN
    AssertEquals_UDINT(
        Expected := E_CommandResult.Aborted,
        Actual := iTestCommand.P_CommandStatus.Result,
        Message := 'Interlock loss handled as abort operation'
    );
ELSE
    AssertTrue(
        Condition := FALSE,
        Message := 'SAFETY CRITICAL: No error indication detected after interlock loss'
    );
END_IF

// If command transitioned to Complete state, let it auto-reset to Idle
IF iTestCommand.P_CommandStatus.StepState = E_CommandState.Complete THEN
    iTestCommand.CyclicLogic();
    AssertEquals_UDINT(
        Expected := E_CommandState.Idle,
        Actual := iTestCommand.P_CommandStatus.StepState,
        Message := 'Command should auto-reset to Idle after completing error handling'
    );
END_IF

TEST_FINISHED();
END_METHOD

METHOD PRIVATE TEST_InterlockLost_SetsCorrectResult
VAR
	TestIdx : DINT := INDEX_INTERLOCKLOST_SETSCORRECTRESULT;
END_VAR
TEST(__POUNAME());

// Initialize test objects - Use index 99 to avoid conflicts
TestCommand[TestIdx].Initialize();
TestComponent[TestIdx].Initialize();
TestCommandConfig[TestIdx].Initialize();
TestPermIntlk[TestIdx].Initialize();

// Safe interface assignments using __QUERYINTERFACE for validation
iTestCommand := TestCommand[TestIdx];

iTestCommandConfig := TestCommandConfig[TestIdx];

iTestComponent := TestComponent[TestIdx];

iTestPermIntlkConfig := TestPermIntlk[TestIdx];

// Interface validation
IF iTestCommand = 0 THEN
    AssertTrue(Condition := FALSE, Message := 'TEST FAILED: iTestCommand interface is null');
    RETURN;
END_IF

// Configure logging to prevent page faults in _ResolveCommandConfiguration()
iTestCommandConfig.P_CommandConfiguration.CommandDescription := 'Test Interlock Lost Result';
IF __ISVALIDREF(iTestCommandConfig.P_CommandConfiguration.BaseConfiguration) THEN
    iTestCommandConfig.P_CommandConfiguration.BaseConfiguration.LogTraceConfiguration.When := E_LogTraceWhen.xRunOnInitOnly;
END_IF
iTestCommandConfig.P_CommandConfiguration.PermIntlkConfiguredAsInterlock := TRUE;
iTestCommandConfig.P_CommandConfiguration.AbortOnInterlockDrop := TRUE;

// Set up initial interlock condition as OK
iTestPermIntlkConfig.P_PermIntlkConfiguration.PermIntlkObj[0].Description := 'Test interlock';
iTestPermIntlkConfig.P_PermIntlkConfiguration.PermIntlkObj[0].Condition := TRUE;
iTestPermIntlkConfig.P_PermIntlkConfiguration.PermIntlkObj[0].Index := 0;
iTestPermIntlkConfig.P_PermIntlkConfiguration.PermIntlkObj[0].Description := 'Test interlock for result verification';

// Setup command with configurations
iTestCommand.InjectConfigurations(
    iComponent := iTestComponent,
    iCommandConfiguration := iTestCommandConfig,
    iPermIntlkConfiguration := iTestPermIntlkConfig
);

// Start execution and get to a state where interlock loss matters
iTestCommand.Execute();
iTestCommand.CyclicLogic(); // Should transition to Execute state

// Verify command is executing before simulating interlock loss
AssertTrue(
    Condition := iTestCommand.P_CommandStatus.StepState <> E_CommandState.Idle,
    Message := 'Command should be executing before testing interlock loss'
);

// Simulate interlock lost by changing the condition
iTestPermIntlkConfig.P_PermIntlkConfiguration.PermIntlkObj[0].Condition := FALSE;

// Process the interlock loss
iTestCommand.CyclicLogic();

// Verify appropriate error response - the specific result depends on implementation
// but some error indication should be present
IF iTestCommand.P_CommandStatus.Result = E_CommandResult.InterlockLost THEN
    AssertEquals_UDINT(
        Expected := E_CommandResult.InterlockLost,
        Actual := iTestCommand.P_CommandStatus.Result,
        Message := 'Command correctly sets InterlockLost result'
    );
    // Policy: InterlockLost must set Error=TRUE
    AssertTrue(
        Condition := iTestCommand.P_CommandStatus.BaseStatus.Error,
        Message := 'POLICY REQUIREMENT: InterlockLost must set Error=TRUE'
    );
ELSIF iTestCommand.P_CommandStatus.Result = E_CommandResult.Aborted THEN
    AssertEquals_UDINT(
        Expected := E_CommandResult.Aborted,
        Actual := iTestCommand.P_CommandStatus.Result,
        Message := 'Command handles interlock loss as abort'
    );
ELSIF iTestCommand.P_CommandStatus.BaseStatus.Error THEN
    AssertTrue(
        Condition := TRUE,
        Message := 'Command indicates interlock loss through Error flag'
    );
ELSE
    AssertTrue(
        Condition := FALSE,
        Message := 'SAFETY CRITICAL: Command must indicate interlock loss through result or error flag'
    );
END_IF

// Verify command stops execution when interlock is lost
AssertFalse(
    Condition := iTestCommand.P_CommandStatus.BaseStatus.Busy,
    Message := 'SAFETY CRITICAL: Command must stop when interlock is lost'
);

TEST_FINISHED();
END_METHOD

METHOD PRIVATE TEST_TimerCompletionTime_SetOnCommandComplete
VAR
	TestIdx : DINT := INDEX_TIMERCOMPLETIONTIME_SETONCOMMANDCOMPLETE;
	completionTimeBefore : ULINT;
	completionTimeAfter : ULINT;
	triggerTime : ULINT;
END_VAR
TEST(__POUNAME());

// Purpose: Verify LastCommandCompletionTime is set accurately when command completes
// Impact: Ensures elapsed time calculations include proper completion timestamp

// Initialize test objects
TestCommand[TestIdx].Initialize();
TestComponent[TestIdx].Initialize();
TestCommandConfig[TestIdx].Initialize();

// Safe interface assignments
iTestCommand := TestCommand[TestIdx];

iTestCommandConfig := TestCommandConfig[TestIdx];

iTestComponent := TestComponent[TestIdx];

iTestPermIntlkConfig := TestCommandConfig[TestIdx];

// Interface validation
IF iTestCommand = 0 THEN
	AssertTrue(Condition := FALSE, Message := 'TEST FAILED: iTestCommand interface is null');
	RETURN;
END_IF

IF iTestCommandConfig = 0 THEN
	AssertTrue(Condition := FALSE, Message := 'TEST FAILED: iTestCommandConfig interface is null');
	RETURN;
END_IF

// Configure command
iTestCommandConfig.P_CommandConfiguration.CommandDescription := 'Timer Completion Test';
iTestCommandConfig.P_CommandConfiguration.TimeoutTime := T#30S;
IF __ISVALIDREF(iTestCommandConfig.P_CommandConfiguration.BaseConfiguration) THEN
    iTestCommandConfig.P_CommandConfiguration.BaseConfiguration.LogTraceConfiguration.When := E_LogTraceWhen.xRunOnInitOnly;
END_IF

// Configure permissive for successful execution
IF iTestPermIntlkConfig <> 0 THEN
	iTestPermIntlkConfig.P_PermIntlkConfiguration.PermIntlkObj[1].Description := 'Timer Completion Test Permissive';
	iTestPermIntlkConfig.P_PermIntlkConfiguration.PermIntlkObj[1].Condition := TRUE;
END_IF

// Setup command with configurations
iTestCommand.InjectConfigurations(
	iComponent := iTestComponent,
	iCommandConfiguration := iTestCommandConfig,
	iPermIntlkConfiguration := iTestPermIntlkConfig
);

// Verify initial state - completion time should be zero
AssertEquals_ULINT(
	Expected := 0,
	Actual := iTestCommand.P_CommandStatus.LastCommandCompletionTime,
	Message := 'Initial completion time should be zero'
);

// Start and run command through completion
iTestCommand.Execute();
iTestCommand.CyclicLogic(); // Execute state
iTestCommand.CyclicLogic(); // Monitor state

// Record time before completion
completionTimeBefore := Tc2_System.F_GetSystemTime();

// Complete the command - this should set completion time
iTestCommand.CyclicLogic(); // Complete state

// Record time after completion
completionTimeAfter := Tc2_System.F_GetSystemTime();

// Verify completion time was set and is within reasonable bounds
AssertTrue(
	Condition := iTestCommand.P_CommandStatus.LastCommandCompletionTime > 0,
	Message := 'LastCommandCompletionTime should be set after completion'
);

AssertTrue(
	Condition := iTestCommand.P_CommandStatus.LastCommandCompletionTime >= completionTimeBefore,
	Message := 'LastCommandCompletionTime should be >= time before completion'
);

AssertTrue(
	Condition := iTestCommand.P_CommandStatus.LastCommandCompletionTime <= completionTimeAfter,
	Message := 'LastCommandCompletionTime should be <= time after completion'
);

// Verify completion time is after trigger time
triggerTime := iTestCommand.P_CommandStatus.LastCommandTriggerTime;
AssertTrue(
	Condition := iTestCommand.P_CommandStatus.LastCommandCompletionTime >= triggerTime,
	Message := 'LastCommandCompletionTime should be >= LastCommandTriggerTime'
);

// Verify elapsed time is calculated correctly
AssertTrue(
	Condition := iTestCommand.P_CommandStatus.LastCommandElapsedTime > LTIME#0s,
	Message := 'LastCommandElapsedTime should be > 0 after completion'
);

TEST_FINISHED();
END_METHOD

METHOD PRIVATE TEST_TimerIntegration_WithCommandStateMachine
VAR
	TestIdx : DINT := INDEX_TIMERINTEGRATION_WITHCOMMANDSTATEMACHINE;
	elapsedInExecute : LTIME;
	elapsedInMonitor : LTIME;
	elapsedInComplete : LTIME;
END_VAR
TEST(__POUNAME());

// Purpose: Verify timer integration with FB_Command state machine transitions
// Impact: Ensures timer behavior aligns correctly with command lifecycle

// Initialize test objects
TestCommand[TestIdx].Initialize();
TestComponent[TestIdx].Initialize();
TestCommandConfig[TestIdx].Initialize();

// Safe interface assignments
iTestCommand := TestCommand[TestIdx];

iTestCommandConfig := TestCommandConfig[TestIdx];

iTestComponent := TestComponent[TestIdx];

iTestPermIntlkConfig := TestCommandConfig[TestIdx];

// Interface validation
IF iTestCommand = 0 THEN
	AssertTrue(Condition := FALSE, Message := 'TEST FAILED: iTestCommand interface is null');
	RETURN;
END_IF

IF iTestCommandConfig = 0 THEN
	AssertTrue(Condition := FALSE, Message := 'TEST FAILED: iTestCommandConfig interface is null');
	RETURN;
END_IF

// Configure command
iTestCommandConfig.P_CommandConfiguration.CommandDescription := 'Timer State Integration Test';
iTestCommandConfig.P_CommandConfiguration.TimeoutTime := T#30S;
IF __ISVALIDREF(iTestCommandConfig.P_CommandConfiguration.BaseConfiguration) THEN
    iTestCommandConfig.P_CommandConfiguration.BaseConfiguration.LogTraceConfiguration.When := E_LogTraceWhen.xRunOnInitOnly;
END_IF

// Configure permissive for successful execution
IF iTestPermIntlkConfig <> 0 THEN
	iTestPermIntlkConfig.P_PermIntlkConfiguration.PermIntlkObj[1].Description := 'Timer Integration Test Permissive';
	iTestPermIntlkConfig.P_PermIntlkConfiguration.PermIntlkObj[1].Condition := TRUE;
END_IF

// Setup command with configurations
iTestCommand.InjectConfigurations(
	iComponent := iTestComponent,
	iCommandConfiguration := iTestCommandConfig,
	iPermIntlkConfiguration := iTestPermIntlkConfig
);

// Verify initial state - timer should not be running
AssertEquals_UDINT(
	Expected := E_CommandState.Idle,
	Actual := iTestCommand.P_CommandStatus.StepState,
	Message := 'Initial state should be Idle'
);

AssertEquals_LTIME(
	Expected := LTIME#0s,
	Actual := iTestCommand.P_CommandStatus.LastCommandElapsedTime,
	Message := 'Initial elapsed time should be 0'
);

// Start execution - timer should start
iTestCommand.Execute();

// Verify Idle → Execute transition and timer start
AssertTrue(
	Condition := iTestCommand.P_CommandStatus.BaseStatus.Busy,
	Message := 'Command should be Busy after Execute()'
);

AssertTrue(
	Condition := iTestCommand.P_CommandStatus.LastCommandTriggerTime > 0,
	Message := 'Timer should start when command becomes Busy'
);

// Progress to Execute state
iTestCommand.CyclicLogic(); // Execute state

AssertEquals_UDINT(
	Expected := E_CommandState.Execute,
	Actual := iTestCommand.P_CommandStatus.StepState,
	Message := 'Command should be in Execute state'
);

elapsedInExecute := iTestCommand.P_CommandStatus.LastCommandElapsedTime;
AssertTrue(
	Condition := elapsedInExecute >= LTIME#0s,
	Message := 'Elapsed time should be >= 0 in Execute state'
);

// Progress to Monitor state
iTestCommand.CyclicLogic(); // Monitor state

AssertEquals_UDINT(
	Expected := E_CommandState.Monitor,
	Actual := iTestCommand.P_CommandStatus.StepState,
	Message := 'Command should be in Monitor state'
);

elapsedInMonitor := iTestCommand.P_CommandStatus.LastCommandElapsedTime;
AssertTrue(
	Condition := elapsedInMonitor >= elapsedInExecute,
	Message := 'Elapsed time should continue increasing in Monitor state'
);

// Progress to Complete state
iTestCommand.CyclicLogic(); // Complete state

AssertEquals_UDINT(
	Expected := E_CommandState.Complete,
	Actual := iTestCommand.P_CommandStatus.StepState,
	Message := 'Command should be in Complete state'
);

elapsedInComplete := iTestCommand.P_CommandStatus.LastCommandElapsedTime;
AssertTrue(
	Condition := elapsedInComplete >= elapsedInMonitor,
	Message := 'Elapsed time should be finalized in Complete state'
);

// Verify timer stopped when command completed
AssertFalse(
	Condition := iTestCommand.P_CommandStatus.BaseStatus.Busy,
	Message := 'Timer should stop when command completes (Busy=FALSE)'
);

AssertTrue(
	Condition := iTestCommand.P_CommandStatus.BaseStatus.Done,
	Message := 'Command should show Done=TRUE when completed'
);

// Verify completion time was set
AssertTrue(
	Condition := iTestCommand.P_CommandStatus.LastCommandCompletionTime > 0,
	Message := 'Completion time should be set when command completes'
);

// Verify completion time is after trigger time
AssertTrue(
	Condition := iTestCommand.P_CommandStatus.LastCommandCompletionTime >= iTestCommand.P_CommandStatus.LastCommandTriggerTime,
	Message := 'Completion time should be >= trigger time'
);

TEST_FINISHED();
END_METHOD

METHOD PRIVATE TEST_TimerPauseResume_ElapsedTimeAccuracy
VAR
	TestIdx : DINT := INDEX_TIMERPAUSERESUME_ELAPSEDTIMEACCURACY;
	elapsedBeforePause : LTIME;
	elapsedAfterResume : LTIME;
	elapsedAfterComplete : LTIME;
END_VAR
TEST(__POUNAME());

// Purpose: Verify timer behavior during pause/resume cycles
// Impact: Ensures elapsed time accuracy across pause/resume operations

// Initialize test objects
TestCommand[TestIdx].Initialize();
TestComponent[TestIdx].Initialize();
TestCommandConfig[TestIdx].Initialize();

// Safe interface assignments
iTestCommand := TestCommand[TestIdx];

iTestCommandConfig := TestCommandConfig[TestIdx];

iTestComponent := TestComponent[TestIdx];

iTestPermIntlkConfig := TestCommandConfig[TestIdx];

// Interface validation
IF iTestCommand = 0 THEN
	AssertTrue(Condition := FALSE, Message := 'TEST FAILED: iTestCommand interface is null');
	RETURN;
END_IF

IF iTestCommandConfig = 0 THEN
	AssertTrue(Condition := FALSE, Message := 'TEST FAILED: iTestCommandConfig interface is null');
	RETURN;
END_IF

// Configure command
iTestCommandConfig.P_CommandConfiguration.CommandDescription := 'Timer Pause Resume Test';
iTestCommandConfig.P_CommandConfiguration.TimeoutTime := T#30S;
IF __ISVALIDREF(iTestCommandConfig.P_CommandConfiguration.BaseConfiguration) THEN
    iTestCommandConfig.P_CommandConfiguration.BaseConfiguration.LogTraceConfiguration.When := E_LogTraceWhen.xRunOnInitOnly;
END_IF

// Configure permissive for successful execution
IF iTestPermIntlkConfig <> 0 THEN
	iTestPermIntlkConfig.P_PermIntlkConfiguration.PermIntlkObj[1].Description := 'Timer Pause Test Permissive';
	iTestPermIntlkConfig.P_PermIntlkConfiguration.PermIntlkObj[1].Condition := TRUE;
	iTestPermIntlkConfig.P_PermIntlkConfiguration.PermIntlkObj[1].Index := 1;
	TestPermIntlk[TestIdx].Initialize();
	TestPermIntlk[TestIdx].CyclicLogic(); // Update permissive evaluation
END_IF

// Setup command with configurations
iTestCommand.InjectConfigurations(
	iComponent := iTestComponent,
	iCommandConfiguration := iTestCommandConfig,
	iPermIntlkConfiguration := iTestPermIntlkConfig
);

// Start command execution
iTestCommand.Execute();
iTestCommand.CyclicLogic(); // Execute state
iTestCommand.CyclicLogic(); // Monitor state

// Record elapsed time before pause
elapsedBeforePause := iTestCommand.P_CommandStatus.LastCommandElapsedTime;

// Pause the command
iTestCommand.Pause();

// Verify command is paused
AssertEquals_UDINT(
	Expected := E_CommandState.Paused,
	Actual := iTestCommand.P_CommandStatus.StepState,
	Message := 'Command should be in Paused state'
);

// Run several cycles while paused - elapsed time should not increase significantly
iTestCommand.CyclicLogic();
iTestCommand.CyclicLogic();
iTestCommand.CyclicLogic();

// Resume the command
iTestCommand.Resume();
iTestCommand.CyclicLogic(); // Process resume and return to Monitor state

// Verify command resumed to Monitor state
AssertEquals_UDINT(
	Expected := E_CommandState.Monitor,
	Actual := iTestCommand.P_CommandStatus.StepState,
	Message := 'Command should return to Monitor state after resume'
);

// Record elapsed time after resume
elapsedAfterResume := iTestCommand.P_CommandStatus.LastCommandElapsedTime;

// Complete the command
iTestCommand.Complete(); // Signal completion
iTestCommand.CyclicLogic(); // Complete state

// Record final elapsed time
elapsedAfterComplete := iTestCommand.P_CommandStatus.LastCommandElapsedTime;

// Verify elapsed time progression
AssertTrue(
	Condition := elapsedAfterResume >= elapsedBeforePause,
	Message := 'Elapsed time after resume should be >= elapsed time before pause'
);

AssertTrue(
	Condition := elapsedAfterComplete >= elapsedAfterResume,
	Message := 'Final elapsed time should be >= elapsed time after resume'
);

// Verify timer functionality during pause/resume
AssertTrue(
	Condition := elapsedAfterComplete > LTIME#0s,
	Message := 'Final elapsed time should be > 0 after pause/resume cycle'
);

TEST_FINISHED();
END_METHOD

METHOD PRIVATE TEST_TimerStopsOnCommandComplete_NotTimeout
VAR
	TestIdx : DINT := INDEX_TIMERSTOPSONCOMMANDCOMPLETE_NOTTIMEOUT;
	elapsedAtComplete : LTIME;
	timeoutTime : TIME;
END_VAR
TEST(__POUNAME());

// Purpose: Verify timer stops immediately on successful completion, not on timeout
// Impact: Ensures successful commands don't run full timeout duration

// Initialize test objects
TestCommand[TestIdx].Initialize();
TestComponent[TestIdx].Initialize();
TestCommandConfig[TestIdx].Initialize();

// Safe interface assignments
iTestCommand := TestCommand[TestIdx];

iTestCommandConfig := TestCommandConfig[TestIdx];

iTestComponent := TestComponent[TestIdx];

iTestPermIntlkConfig := TestCommandConfig[TestIdx];

// Interface validation
IF iTestCommand = 0 THEN
	AssertTrue(Condition := FALSE, Message := 'TEST FAILED: iTestCommand interface is null');
	RETURN;
END_IF

IF iTestCommandConfig = 0 THEN
	AssertTrue(Condition := FALSE, Message := 'TEST FAILED: iTestCommandConfig interface is null');
	RETURN;
END_IF

// Configure command with long timeout
timeoutTime := T#30S;
iTestCommandConfig.P_CommandConfiguration.CommandDescription := 'Timer Stop Test';
iTestCommandConfig.P_CommandConfiguration.TimeoutTime := timeoutTime;
IF __ISVALIDREF(iTestCommandConfig.P_CommandConfiguration.BaseConfiguration) THEN
    iTestCommandConfig.P_CommandConfiguration.BaseConfiguration.LogTraceConfiguration.When := E_LogTraceWhen.xRunOnInitOnly;
END_IF

// Configure permissive for successful execution
IF iTestPermIntlkConfig <> 0 THEN
	iTestPermIntlkConfig.P_PermIntlkConfiguration.PermIntlkObj[1].Description := 'Timer Stop Test Permissive';
	iTestPermIntlkConfig.P_PermIntlkConfiguration.PermIntlkObj[1].Condition := TRUE;
END_IF

// Setup command with configurations
iTestCommand.InjectConfigurations(
	iComponent := iTestComponent,
	iCommandConfiguration := iTestCommandConfig,
	iPermIntlkConfiguration := iTestPermIntlkConfig
);

// Execute command to completion
iTestCommand.Execute();
iTestCommand.CyclicLogic(); // Execute state
iTestCommand.CyclicLogic(); // Monitor state
iTestCommand.CyclicLogic(); // Complete state

// Verify command completed successfully
AssertEquals_UDINT(
	Expected := E_CommandState.Complete,
	Actual := iTestCommand.P_CommandStatus.StepState,
	Message := 'Command should be in Complete state'
);

AssertEquals_UDINT(
	Expected := E_CommandResult.Ok,
	Actual := iTestCommand.P_CommandStatus.Result,
	Message := 'Command should have Ok result (not timeout)'
);

// Record elapsed time at completion
elapsedAtComplete := iTestCommand.P_CommandStatus.LastCommandElapsedTime;

// Verify elapsed time is much less than timeout duration
// Successful commands should complete in milliseconds, not seconds
AssertTrue(
	Condition := elapsedAtComplete < TIME_TO_LTIME(timeoutTime),
	Message := 'Elapsed time should be much less than timeout duration for successful completion'
);

// Verify elapsed time is reasonable (should be very short for fast completion)
AssertTrue(
	Condition := elapsedAtComplete < LTIME#1s,
	Message := 'Elapsed time should be < 1s for immediate completion'
);

// Verify timer is no longer running
AssertFalse(
	Condition := iTestCommand.P_CommandStatus.BaseStatus.Busy,
	Message := 'Timer should stop when command completes (Busy=FALSE)'
);

AssertTrue(
	Condition := iTestCommand.P_CommandStatus.BaseStatus.Done,
	Message := 'Command should show Done=TRUE when successfully completed'
);

TEST_FINISHED();
END_METHOD

METHOD PRIVATE TEST_TimerTriggerTime_SetOnCommandStart
VAR
	TestIdx : DINT := INDEX_TIMERPAUSERESUME_ELAPSEDTIMEACCURACY;
	triggerTimeBefore : ULINT;
	triggerTimeAfter : ULINT;
	currentTime : ULINT;
END_VAR
TEST(__POUNAME());

// Purpose: Verify LastCommandTriggerTime is set accurately when timer starts
// Impact: Ensures elapsed time calculations are based on correct start time

// Initialize test objects
TestCommand[TestIdx].Initialize();
TestComponent[TestIdx].Initialize();
TestCommandConfig[TestIdx].Initialize();

// Safe interface assignments using __QUERYINTERFACE for validation
iTestCommand := TestCommand[TestIdx];

iTestCommandConfig := TestCommandConfig[TestIdx];

iTestComponent := TestComponent[TestIdx];

iTestPermIntlkConfig := TestCommandConfig[TestIdx];

// Interface validation
IF iTestCommand = 0 THEN
	AssertTrue(Condition := FALSE, Message := 'TEST FAILED: iTestCommand interface is null');
	RETURN;
END_IF

IF iTestCommandConfig = 0 THEN
	AssertTrue(Condition := FALSE, Message := 'TEST FAILED: iTestCommandConfig interface is null');
	RETURN;
END_IF

// Configure command
iTestCommandConfig.P_CommandConfiguration.CommandDescription := 'Timer Trigger Test';
iTestCommandConfig.P_CommandConfiguration.TimeoutTime := T#30S;
IF __ISVALIDREF(iTestCommandConfig.P_CommandConfiguration.BaseConfiguration) THEN
    iTestCommandConfig.P_CommandConfiguration.BaseConfiguration.LogTraceConfiguration.When := E_LogTraceWhen.xRunOnInitOnly;
END_IF

// Configure permissive for successful execution
IF iTestPermIntlkConfig <> 0 THEN
	iTestPermIntlkConfig.P_PermIntlkConfiguration.PermIntlkObj[1].Description := 'Timer Test Permissive';
	iTestPermIntlkConfig.P_PermIntlkConfiguration.PermIntlkObj[1].Condition := TRUE;
END_IF

// Setup command with configurations
iTestCommand.InjectConfigurations(
	iComponent := iTestComponent,
	iCommandConfiguration := iTestCommandConfig,
	iPermIntlkConfiguration := iTestPermIntlkConfig
);

// Verify initial state - trigger time should be zero
AssertEquals_ULINT(
	Expected := 0,
	Actual := iTestCommand.P_CommandStatus.LastCommandTriggerTime,
	Message := 'Initial trigger time should be zero'
);

// Record time before starting command
triggerTimeBefore := Tc2_System.F_GetSystemTime();

// Start command execution - this should set trigger time
iTestCommand.Execute();

// Record time after starting command
triggerTimeAfter := Tc2_System.F_GetSystemTime();

// Verify trigger time was set and is within reasonable bounds
AssertTrue(
	Condition := iTestCommand.P_CommandStatus.LastCommandTriggerTime > 0,
	Message := 'LastCommandTriggerTime should be set after Execute()'
);

AssertTrue(
	Condition := iTestCommand.P_CommandStatus.LastCommandTriggerTime >= triggerTimeBefore,
	Message := 'LastCommandTriggerTime should be >= time before Execute()'
);

AssertTrue(
	Condition := iTestCommand.P_CommandStatus.LastCommandTriggerTime <= triggerTimeAfter,
	Message := 'LastCommandTriggerTime should be <= time after Execute()'
);

// Run CyclicLogic to advance states
iTestCommand.CyclicLogic(); // Execute state
iTestCommand.CyclicLogic(); // Monitor state

// Verify trigger time remains constant after initial setting
currentTime := iTestCommand.P_CommandStatus.LastCommandTriggerTime;

iTestCommand.CyclicLogic(); // Complete state

AssertEquals_ULINT(
	Expected := currentTime,
	Actual := iTestCommand.P_CommandStatus.LastCommandTriggerTime,
	Message := 'LastCommandTriggerTime should remain constant after initial setting'
);

TEST_FINISHED();
END_METHOD

END_FUNCTION_BLOCK

// Tests/FB_CommandTestsIV
FUNCTION_BLOCK FB_CommandTestsIV EXTENDS TcUnit.FB_TestSuite
VAR CONSTANT
	// Test method index constants - one unique index per test method (0-113)

	// GivenCommand* helper test methods (0-25)
	INDEX_GIVENCOMMAND_WHENCANCEL_EXPECTREMOVEDFROMQUEUE							: DINT := 0;
	INDEX_GIVENCOMMAND_WHENCYCLICLOGICCALLED_EXPECTUPDATED							: DINT := 1;
	INDEX_GIVENCOMMAND_WHENEXECUTECALLED_EXPECTEXECUTION							: DINT := 2;
	INDEX_GIVENCOMMAND_WHENPAUSECALLED_EXPECTCOMMANDPAUSES							: DINT := 3;
	INDEX_GIVENCOMMAND_WHENQUEUECALLED_EXPECTADDEDTOQUEUE							: DINT := 4;
	INDEX_GIVENCOMMAND_WHENRESETCALLED_EXPECTSTATECLEARED							: DINT := 5;
	INDEX_GIVENCOMMAND_WHENRESUMECALLED_EXPECTCOMMANDRESUMES						: DINT := 6;
	INDEX_GIVENCOMMAND_WHENVALIDATECALLED_EXPECTPERMISSIVEOK						: DINT := 7;
	INDEX_GIVENCOMMAND_WHENVALIDATECALLED_EXPECTMATCHCONFIG							: DINT := 8;
	INDEX_GIVENCOMMANDALREADYRUNNING_WHENEXECUTE_CONFLICT							: DINT := 9;
	INDEX_GIVENCOMMANDEXECUTED_WHENCYCLICLOGICRUNS_EXPECTSTATEPROGRESSION			: DINT := 10;
	INDEX_GIVENCOMMANDINIDLESTATE_WHENCANCEL_EXPECTNOACTIONTAKEN					: DINT := 11;
	INDEX_GIVENCOMMANDINVALID_WHENVALIDATECALLED_EXPECTFALSE						: DINT := 12;
	INDEX_GIVENCOMMANDPAUSED_WHENABORT_EXPECTCOMMANDABORTEDANDSTATUSUPDATED			: DINT := 13;
	INDEX_GIVENCOMMANDPAUSED_WHENRESUME_EXPECTCOMMANDRESUMESEXECUTION				: DINT := 14;
	INDEX_GIVENCOMMANDQUEUED_WHENABORT_EXPECTCOMMANDABORTEDANDSTATUSUPDATED			: DINT := 15;
	INDEX_GIVENCOMMANDQUEUED_WHENCANCEL_EXPECTCOMMANDREMOVEDFROMQUEUE				: DINT := 16;
	INDEX_GIVENCOMMANDVALIDATED_WHENVALIDATECALLED_EXPECTTRUE						: DINT := 17;
	INDEX_GIVENCOMPONENTRESET_WHENRESETCALLED_EXPECTALLCOMMANDSTATECLEARED			: DINT := 18;
	INDEX_GIVENINJECTEDCONFIGURATIONSVALID_EXPECTINTERFACESSTOREDANDINITIALIZED		: DINT := 19;
	INDEX_GIVENINVALIDCONFIGURATION_WHENINJECTCONFIGURATIONCALLED_EXPECTINITFAILURE	: DINT := 20;
	INDEX_GIVENINVALIDCONFIGURATIONS_WHENINJECTCONFIGURATIONS_EXPECTINITFAILURE		: DINT := 21;
	INDEX_GIVENRUNNINGCOMMAND_WHENPAUSE_EXPECTCOMMANDTRANSITIONSTOPAUSEDSTATE		: DINT := 22;
	INDEX_GIVENTIMERSTARTED_WHENCYCLICLOGICRUNS_EXPECTELAPSEDTIMEINCREASES			: DINT := 23;
	INDEX_GIVENTIMERSTOPPED_WHENCYCLICLOGICRUNS_EXPECTELAPSEDTIMEREMAINCONSTANT		: DINT := 24;
	INDEX_GIVENVALIDCONFIGURATION_WHENINJECTCONFIGURATIONCALLED_EXPECTCONFIGSTORED	: DINT := 25;

	// TEST_* methods (26-113)
	INDEX_ABORT_AFTERCOMPLETE_IGNOREDWITHWARNING									: DINT := 26;
	INDEX_ABORT_ERRORCLASSIFICATION													: DINT := 27;
	INDEX_ABORT_WHENIDLEQUEUED_SETSRESULTABORTED									: DINT := 28;
	INDEX_ABORTAFTERCOMPLETE_STATEPRESERVATION										: DINT := 29;
	INDEX_ABORTDURINGCOMPLETIONWAIT													: DINT := 30;
	INDEX_ACCEPTEDCOMMAND_WHENEXECUTED_RESULTBECOMESOK								: DINT := 31;
	INDEX_BADREQUEST_INTERLOCKMISCONFIGURED											: DINT := 32;
	INDEX_BUSYCOMMANDELAPSEDTIMEEQUALS_COMMANDABORTED								: DINT := 33;
	INDEX_CANCEL_FROMQUEUEDSTATE													: DINT := 34;
	INDEX_CANCEL_REMOVESCOMMANDFROMQUEUE											: DINT := 35;
	INDEX_CANCEL_SETSCOMMANDSTATUSTOCANCELLED										: DINT := 36;
	INDEX_CANCEL_SETSRESULTCANCELLED												: DINT := 37;
	INDEX_CANCEL_WHENBUSY_REJECTED_NOCHANGETOSTATE									: DINT := 38;
	INDEX_COMMAND_LOCALREFERENCES_INITIALIZEDPROPERLY								: DINT := 39;
	INDEX_COMMAND_MISSINGCONFIGINTERFACE_FALLBACK									: DINT := 40;
	INDEX_COMMAND_PERMINTLKCHILD_INITIALIZED										: DINT := 41;
	INDEX_COMMANDATTEMPTSEXCEEDRETRYCOUNT											: DINT := 42;
	INDEX_COMMANDCOMPLETES_STATUSDONEANDCLEARED										: DINT := 43;
	INDEX_COMMANDSTATUS_CONFIGREF_POINTSTOCONFIGURATION								: DINT := 44;
	INDEX_COMMANDTIMEOUT_TRIGGERSRESET												: DINT := 45;
	INDEX_COMPLETE_ERROR_PERSISTSUNTILRESET											: DINT := 46;
	INDEX_COMPLETE_OK_AUTORESETNEXTCYCLE											: DINT := 47;
	INDEX_COMPLETESTATE_PRESERVESABORTEDRESULT										: DINT := 48;
	INDEX_COMPLETESTATE_PRESERVESTIMEOUTRESULT										: DINT := 49;
	INDEX_COMPLETESTATE_SETSOKFORSUCCESSFUL											: DINT := 50;
	INDEX_COMPLETIONCALLBACKTOSEQUENCER												: DINT := 51;
	INDEX_COMPLETIONCONDITIONEVALUATION												: DINT := 52;
	INDEX_COMPLETIONCONDITIONWITHTIMEOUT											: DINT := 53;
	INDEX_COMPLETIONWITHINTERLOCKDROP												: DINT := 54;
	INDEX_COMPLEXCOMPLETIONCONDITION												: DINT := 55;
	INDEX_COMPONENTBUSY_DURINGVALIDATION_RESULTCONFLICT								: DINT := 56;
	INDEX_CONFIG_FALLBACKTOLOCAL_WHENINJECTEDINVALID								: DINT := 57;
	INDEX_CONFIG_RECOVERYTOINJECTED_WHENVALIDAGAIN									: DINT := 58;
	INDEX_CONFIGURATIONRESOLUTION_HANDLESVALIDINVALID								: DINT := 59;
	INDEX_CYCLICLOGIC_STATEMACHINEPROGRESSION										: DINT := 60;
	INDEX_DISCRETECOMPLETIONCONDITION												: DINT := 61;
	INDEX_DYNAMICCOMPLETIONCONDITIONUPDATE											: DINT := 62;
	INDEX_EDGETRIGGERED_STATEMACHINEEXECUTION										: DINT := 63;
	INDEX_EXECUTE_HAPPYPATH_TRANSITIONSTOMONITOR									: DINT := 64;
	INDEX_EXECUTE_STATEMACHINEPROGRESSION											: DINT := 65;
	INDEX_EXECUTE_TRANSITIONSFROMACCEPTEDTOOK										: DINT := 66;
	INDEX_EXECUTE_VALIDATESBEFOREACCEPTING											: DINT := 67;
	INDEX_EXECUTE_WHENPERMISSIVEMISSING_RETURNSFORBIDDEN							: DINT := 68;
	INDEX_FASTCOMPLETIONINONESCAN													: DINT := 69;
	INDEX_FORBIDDEN_RESUMEWITHOUTPERMISSIVE											: DINT := 70;
	INDEX_INJECTCONFIGURATIONS_STORESINTERFACES										: DINT := 71;
	INDEX_INTERFACEINJECTIONCONFIGURATIONRESOLUTION									: DINT := 72;
	INDEX_INTERLOCKDROP_ABORTSCOMMANDWHENCONFIGURED									: DINT := 73;
	INDEX_INTERLOCKDROP_FROMMONITORSTATE											: DINT := 74;
	INDEX_INTERLOCKINVALIDCONFIG_DURINGVALIDATION									: DINT := 75;
	INDEX_INTERLOCKLOST_COMPREHENSIVESTATETRANSITIONS								: DINT := 76;
	INDEX_INTERLOCKLOST_FROMEXECUTESTATE											: DINT := 77;
	INDEX_INTERLOCKLOST_SETSCORRECTRESULT											: DINT := 78;
	INDEX_INTERLOCKREFERENCELOST_DURINGEXECUTION									: DINT := 79;
	INDEX_METHODENABLEMENT_BUSYSTATE_ALLOWABORT										: DINT := 80;
	INDEX_METHODENABLEMENT_DONESTATE_ALLOWRESET										: DINT := 81;
	INDEX_METHODENABLEMENT_IDLEWITHINTERLOK_ALLOWEXECUTE							: DINT := 82;
	INDEX_METHODENABLEMENT_IDLEWITHOUTINTERLOK_REJECT								: DINT := 83;
	INDEX_MOTIONCOMPLETIONCONDITION													: DINT := 84;
	INDEX_OPERATIONTOCOMMANDTRANSLATION												: DINT := 85;
	INDEX_OPERATORABORT_VSINTERLOCKABORT_DIFFERENTRESULTS							: DINT := 86;
	INDEX_PAUSERESUME_STATETRANSITIONS												: DINT := 87;
	INDEX_PAUSERESUMEWITHCOMPLETIONCONDITION										: DINT := 88;
	INDEX_PERMINTLKLOST_DURINGBUSY_COMMANDABORTED									: DINT := 89;
	INDEX_PERMISSIVEFALSE_DURINGVALIDATION_FORBIDDEN								: DINT := 90;
	INDEX_QUEUEOPERATIONS_MULTIPLECOMMANDSATOMICITY									: DINT := 91;
	INDEX_RECIPEMANAGERPROVIDESCOMMANDCONFIG										: DINT := 92;
	INDEX_RESET_CLEARSCOMMANDSTATE													: DINT := 93;
	INDEX_RESULTPERSISTENCE_TERMINALSTATES											: DINT := 94;
	INDEX_RETRYCOUNT_INCREMENTONEXECUTIONSTARTONLY									: DINT := 95;
	INDEX_RUNTIMECOMMANDCONFIGLOSS_INJECTEDREFSINVALIDATED							: DINT := 96;
	INDEX_RUNTIMECOMMANDCONFIGRECOVERY_VALIDREFSRESTORED							: DINT := 97;
	INDEX_SLOWCOMPLETIONMULTIPLESCANS												: DINT := 98;
	INDEX_STEPSTATE_TRANSITIONSANDVALIDATION										: DINT := 99;
	INDEX_SYSTEMATICSTATEVALIDATION_IDLESTATES										: DINT := 100;
	INDEX_SYSTEMATICSTATEVALIDATION_TERMINALSTATES									: DINT := 101;
	INDEX_TERMINALRESULTS_ERRORFLAGCONSISTENCY										: DINT := 102;
	INDEX_TIMEBASEDCOMPLETIONCONDITION												: DINT := 103;
	INDEX_TIMEOUTANDINTERLOCKLOST_SAMECYCLE_PRIORITIZE								: DINT := 104;
	INDEX_TIMERCOMPLETIONTIME_SETONCOMMANDCOMPLETE									: DINT := 105;
	INDEX_TIMERINTEGRATION_WITHCOMMANDSTATEMACHINE									: DINT := 106;
	INDEX_TIMERPAUSERESUME_ELAPSEDTIMEACCURACY										: DINT := 107;
	INDEX_TIMERSTOPSONCOMMANDCOMPLETE_NOTTIMEOUT									: DINT := 108;
	INDEX_TIMERTRIGGERTIME_SETONCOMMANDSTART										: DINT := 109;
	INDEX_VALIDATE_RETURNSPROPERRESULT												: DINT := 110;
	INDEX_VALIDATE_WITHCONTINUOUSEVALUATION											: DINT := 111;
	INDEX_VALIDATIONOK_INTERLOCKDROP_DURINGEXECUTION								: DINT := 112;
	INDEX_VALIDCOMMAND_EXPECTEXECUTED												: DINT := 113;

	// Additional indices for multi-scenario tests
	INDEX_TERMINALRESULTS_CLEANCANCEL												: DINT := 114;
	INDEX_TERMINALRESULTS_INTERLOCKLOST											: DINT := 115;
	INDEX_TERMINALRESULTS_TIMEOUT													: DINT := 116;
	INDEX_TERMINALRESULTS_COMPLETE_OK												: DINT := 117;
	INDEX_TERMINALRESULTS_COMPLETE_ERROR											: DINT := 118;
	INDEX_VALIDATIONOK_INTERLOCKDROP_SCENARIO2										: DINT := 119;

	// Fixed duplicate indices - these tests were incorrectly reusing other test indices
	INDEX_TIMEOUTANDINTERLOCKLOST_SAMECYCLE_PRIORITIZEINTERLOCKLOST					: DINT := 120;
	INDEX_VALIDATE_RETURNSPROPERRESULTBASEDONPERMISSIVES							: DINT := 121;
	INDEX_VALIDATE_WITHCONTINUOUSEVALUATION_PROPER									: DINT := 122;
	INDEX_VALIDATIONOK_INTERLOCKDROPDURINGEXECUTION									: DINT := 123;
	INDEX_VALIDCOMMAND_EXPECTEXECUTED_PROPER										: DINT := 124;
END_VAR

VAR

	// Mock component for testing
	MockComponent 			: FB_ComponentDerivative;

	// Common test interfaces for all methods (FB-level for stability)
	// Initialized to 0 to prevent page faults - will be set by each test method safely
	iTestCommand 			: I_CommandUnderTest;
	iTestCommandConfig 		: I_CommandConfiguration;
	iTestComponent 			: I_ComponentFull;
	iTestPermIntlkConfig 	: I_PermIntlkConfiguration;
	iTestPermIntlk 			: I_PermIntlk;
	iTestPermIntlkEval		: I_PermIntlk;
	
	// Array instances for test methods (indices 0-17)
	TestCommand : ARRAY[GC_Test.INDEX_TestFB_Command_MIN..GC_Test.INDEX_TestFB_Command_MAX] OF FB_CommandUnderTest;
	TestComponent : ARRAY[GC_Test.INDEX_TestFB_Command_MIN..GC_Test.INDEX_TestFB_Command_MAX] OF FB_ComponentDerivative;
	TestCommandConfig : ARRAY[GC_Test.INDEX_TestFB_Command_MIN..GC_Test.INDEX_TestFB_Command_MAX] OF FB_CmdPermIntlkConfiguration;
	TestPermIntlk : ARRAY[GC_Test.INDEX_TestFB_Command_MIN..GC_Test.INDEX_TestFB_Command_MAX] OF FB_PermIntlkCommand;
	MockQueue : ARRAY[GC_Test.INDEX_TestFB_Command_MIN..GC_Test.INDEX_TestFB_Command_MAX] OF FB_RingBufferICmd;
	CommandTimer : ARRAY[GC_Test.INDEX_TestFB_Command_MIN..GC_Test.INDEX_TestFB_Command_MAX] OF FB_CommandElapsedTimer;
//	FileHandler : ARRAY[GC_Test.INDEX_TestFB_Command_MIN..GC_Test.INDEX_TestFB_Command_MAX] OF FB_FileHandlerCsv;
END_VAR

// === Missing Command Tests ===
TEST_Abort_ErrorClassification();
TEST_AcceptedCommand_WhenExecuted_ResultBecomesOk();
TEST_BadRequest_InterlockMisconfigured_ReturnsBadRequest();
TEST_BusyCommandElapsedTimeEqualsTimeout_CommandAborted();
TEST_Cancel_RemovesCommandFromQueue();
TEST_Cancel_SetsCommandStatusToCancelled();
TEST_Cancel_SetsResultToCancelled();
TEST_Command_LocalReferences_InitializedProperly();
TEST_Command_MissingConfigInterface_FallbackToLocal();
TEST_Command_PermIntlkChild_Initialized();
TEST_CommandStatus_ConfigRef_PointsToConfiguration();

METHOD PRIVATE TEST_Abort_ErrorClassification
VAR
	TestIdx : DINT := INDEX_ABORT_ERRORCLASSIFICATION;
	stCommandStatus : ST_CommandStatus;
	stBaseStatus : ST_BaseStatus;
END_VAR
TEST(__POUNAME());

// Policy Decision: "aborted is a terminal state; error flag is a separate bit (in base status)"
// Test verifies that Abort sets Result=Aborted AND Error flag correctly based on abort reason

// Setup test using helper functions
IF NOT GivenValidCommand(
    testIndex := 22,
    TestCommand := TestCommand,
    TestComponent := TestComponent,
    TestCommandConfig := TestCommandConfig,
    iTestCommand := iTestCommand,
    iTestCommandConfig := iTestCommandConfig,
    iTestComponent := iTestComponent,
    iTestPermIntlkConfig := iTestPermIntlkConfig
) THEN
    AssertTrue(FALSE, 'Failed to setup valid command for test');
    RETURN;
END_IF

// Test 1: User-initiated abort (should be terminal state with error flag per implementation)
// Execute command and advance to Monitor state
iTestCommand.Execute();
iTestCommand.CyclicLogic(); // Idle -> Execute
iTestCommand.CyclicLogic(); // Execute -> Monitor

// Verify in Monitor state
AssertEquals_UDINT(
    Expected := E_CommandState.Monitor,
    Actual := iTestCommand.P_CommandStatus.StepState,
    Message := 'Command should be in Monitor state before user abort'
);

// User-initiated abort
iTestCommand.Abort();

// Verify abort result and that error flag matches abort reason
AssertEquals_UDINT(
    Expected := E_CommandResult.Aborted,
    Actual := iTestCommand.P_CommandStatus.Result,
    Message := 'User-initiated abort should set Result to Aborted'
);

// Policy: Aborted should have Error=FALSE (operator/system abort without fault)
AssertFalse(
    Condition := iTestCommand.P_CommandStatus.BaseStatus.Error,
    Message := 'POLICY REQUIREMENT: Aborted should have Error=FALSE per policy'
);

AssertEquals_UDINT(
    Expected := E_CommandState.Idle,
    Actual := iTestCommand.P_CommandStatus.StepState,
    Message := 'Aborted command should return to Idle state'
);

// Test 2: Verify Reset clears both Result and Error flag
iTestCommand.Reset();

AssertEquals_UDINT(
    Expected := E_CommandResult.None,
    Actual := iTestCommand.P_CommandStatus.Result,
    Message := 'Reset should clear Result to None'
);

AssertFalse(
    Condition := iTestCommand.P_CommandStatus.BaseStatus.Error,
    Message := 'Reset should clear Error flag'
);

// Test 3: Verify Aborted state persistence (until Reset)
// Setup fresh command
IF NOT GivenValidCommand(
    testIndex := 23,
    TestCommand := TestCommand,
    TestComponent := TestComponent,
    TestCommandConfig := TestCommandConfig,
    iTestCommand := iTestCommand,
    iTestCommandConfig := iTestCommandConfig,
    iTestComponent := iTestComponent,
    iTestPermIntlkConfig := iTestPermIntlkConfig
) THEN
    AssertTrue(FALSE, 'Failed to setup second command for persistence test');
    RETURN;
END_IF

iTestCommand.Execute();
iTestCommand.CyclicLogic(); // Execute
iTestCommand.Abort();

// Verify Result persists across CyclicLogic calls (per policy decision)
iTestCommand.CyclicLogic();
AssertEquals_UDINT(
    Expected := E_CommandResult.Aborted,
    Actual := iTestCommand.P_CommandStatus.Result,
    Message := 'Aborted result should persist until explicit Reset'
);

TEST_FINISHED();
END_METHOD

METHOD PRIVATE TEST_Cancel_RemovesCommandFromQueue
VAR
	TestIdx : DINT := INDEX_CANCEL_REMOVESCOMMANDFROMQUEUE;
	stCommandStatus : ST_CommandStatus;
	stBaseStatus : ST_BaseStatus;
	stCommandConfiguration : ST_CommandConfiguration;
	MockQueueEntry : ST_SystimeICmd;
	QueueSizeBeforeCancel : ULINT;
	QueueSizeAfterCancel : ULINT;
END_VAR
TEST(__POUNAME());

// Initialize reference objects for stCommandStatus
stCommandStatus.BaseStatus REF= stBaseStatus;
stCommandStatus.ConfigRef REF= stCommandConfiguration;

// Initialize test objects first
TestCommand[TestIdx].Initialize();
TestComponent[TestIdx].Initialize();
TestCommandConfig[TestIdx].Initialize();
MockQueue[TestIdx].Initialize();

// Direct interface assignments
iTestCommand := TestCommand[TestIdx];
iTestCommandConfig := TestCommandConfig[TestIdx];
iTestComponent := TestComponent[TestIdx];

// Configure the command
TestCommandConfig[TestIdx].P_CommandConfiguration.CommandDescription := 'Test Command for Cancel';
IF __ISVALIDREF(TestCommandConfig[TestIdx].P_CommandConfiguration.BaseConfiguration) THEN
    TestCommandConfig[TestIdx].P_CommandConfiguration.BaseConfiguration.LogTraceConfiguration.When := E_LogTraceWhen.xRunOnInitOnly;
END_IF

// Setup command with configurations
iTestCommand.InjectConfigurations(
	iComponent := iTestComponent,
	iCommandConfiguration := iTestCommandConfig,
	iPermIntlkConfiguration := iTestPermIntlkConfig
);

// Test 1: Cancel command that is queued - should remove from queue and set Cancelled result
stBaseStatus.Busy := FALSE;
stBaseStatus.Done := FALSE;
stCommandStatus.BaseStatus REF= stBaseStatus;
IF iTestCommandConfig <> 0 THEN
	stCommandConfiguration := iTestCommandConfig.P_CommandConfiguration;
END_IF
stCommandStatus.StepState := E_CommandState.Idle;
stCommandStatus.Result := E_CommandResult.Accepted;
iTestCommand.SetCommandStatus(stCommandStatus);

// Add command to component's queue
MockQueueEntry.iCmd := iTestCommand;
MockQueueEntry.systimestamp := 0;
iTestComponent.P_CommandQueue.AddObject(RefObject := MockQueueEntry);

// Get queue size before cancel
QueueSizeBeforeCancel := iTestComponent.P_CommandQueue.P_RingBufferStatus.ObjectCountInBufferPrim;

// Verify command is in queued state before cancel
AssertEquals_UDINT(
	Expected := E_CommandState.Idle,
	Actual := iTestCommand.P_CommandStatus.StepState,
	Message := 'Command should be in Queued state before cancel'
);

// Cancel the command - should remove it from queue
iTestCommand.Cancel();

// Get queue size after cancel
QueueSizeAfterCancel := iTestComponent.P_CommandQueue.P_RingBufferStatus.ObjectCountInBufferPrim;

// Verify command was removed from queue
AssertTrue(
	Condition := QueueSizeAfterCancel < QueueSizeBeforeCancel,
	Message := 'Queue size should decrease after cancelling queued command'
);

// Verify command result is set to Cancelled
AssertEquals_UDINT(
	Expected := E_CommandResult.Cancelled,
	Actual := iTestCommand.P_CommandStatus.Result,
	Message := 'Command result should be Cancelled after calling Cancel()'
);

// Test 2: Cancel command from Executing state - should not affect queue but set Cancelled result
stBaseStatus.Busy := TRUE;
stBaseStatus.Done := FALSE;
stCommandStatus.BaseStatus REF= stBaseStatus;
IF iTestCommandConfig <> 0 THEN
	stCommandConfiguration := iTestCommandConfig.P_CommandConfiguration;
END_IF
stCommandStatus.StepState := E_CommandState.Execute;
stCommandStatus.Result := E_CommandResult.Accepted;
iTestCommand.SetCommandStatus(stCommandStatus);

iTestCommand.Cancel();

// Cancel from executing state should be ignored - result should remain unchanged
AssertEquals_UDINT(
	Expected := E_CommandResult.Accepted,
	Actual := iTestCommand.P_CommandStatus.Result,
	Message := 'Cancel during execution should be ignored - result remains Accepted'
);

// Test 3: Cancel command from Paused state - should be ignored (Paused commands are Busy=TRUE)
stBaseStatus.Busy := TRUE;
stBaseStatus.Done := FALSE;
stCommandStatus.BaseStatus REF= stBaseStatus;
IF iTestCommandConfig <> 0 THEN
	stCommandConfiguration := iTestCommandConfig.P_CommandConfiguration;
END_IF
stCommandStatus.StepState := E_CommandState.Paused;
stCommandStatus.Result := E_CommandResult.Accepted;
iTestCommand.SetCommandStatus(stCommandStatus);

iTestCommand.Cancel();

AssertEquals_UDINT(
	Expected := E_CommandResult.Accepted,
	Actual := iTestCommand.P_CommandStatus.Result,
	Message := 'Cancel should be ignored for Paused commands (Busy=TRUE) - result remains Accepted'
);

// Test 4: Cancel when command not in queue should not cause errors but still set result
stBaseStatus.Busy := FALSE;
stBaseStatus.Done := FALSE;
stCommandStatus.BaseStatus REF= stBaseStatus;
IF iTestCommandConfig <> 0 THEN
	stCommandConfiguration := iTestCommandConfig.P_CommandConfiguration;
END_IF
stCommandStatus.StepState := E_CommandState.Idle;
stCommandStatus.Result := E_CommandResult.None;
iTestCommand.SetCommandStatus(stCommandStatus);

iTestCommand.Cancel();

// Should not crash and should still set Cancelled result
AssertEquals_UDINT(
	Expected := E_CommandResult.Cancelled,
	Actual := iTestCommand.P_CommandStatus.Result,
	Message := 'Cancel should set Cancelled result even when command not in queue'
);

TEST_FINISHED();
END_METHOD

METHOD PRIVATE TEST_Cancel_SetsCommandStatusToCancelled
VAR
	TestIdx : DINT := INDEX_CANCEL_SETSCOMMANDSTATUSTOCANCELLED;
	stCommandStatus : ST_CommandStatus;
	stBaseStatus : ST_BaseStatus;
	stCommandConfiguration : ST_CommandConfiguration;
END_VAR
TEST(__POUNAME());

// Initialize reference objects for stCommandStatus
stCommandStatus.BaseStatus REF= stBaseStatus;
stCommandStatus.ConfigRef REF= stCommandConfiguration;

// Initialize test objects first
TestCommand[TestIdx].Initialize();
TestComponent[TestIdx].Initialize();
TestCommandConfig[TestIdx].Initialize();

// Safe interface assignments using __QUERYINTERFACE for validation
iTestCommand := TestCommand[TestIdx];

iTestCommandConfig := TestCommandConfig[TestIdx];

iTestComponent := TestComponent[TestIdx];

iTestPermIntlkConfig := TestCommandConfig[TestIdx];

// Configure the command
TestCommandConfig[TestIdx].P_CommandConfiguration.CommandDescription := 'Test Command for Cancel';
IF __ISVALIDREF(TestCommandConfig[TestIdx].P_CommandConfiguration.BaseConfiguration) THEN
    TestCommandConfig[TestIdx].P_CommandConfiguration.BaseConfiguration.LogTraceConfiguration.When := E_LogTraceWhen.xRunOnInitOnly;
END_IF

// Configure permissive to be OK for successful validation
IF iTestPermIntlkConfig <> 0 THEN
	iTestPermIntlkConfig.P_PermIntlkConfiguration.PermIntlkObj[1].Description := 'Test Permissive';
	iTestPermIntlkConfig.P_PermIntlkConfiguration.PermIntlkObj[1].Condition := TRUE;
	iTestPermIntlkConfig.P_PermIntlkConfiguration.PermIntlkObj[1].Index := 1;
END_IF

// Interface validation with protection
IF iTestCommand = 0 THEN
	AssertTrue(Condition := FALSE, Message := 'TEST FAILED: iTestCommand interface is null - cannot execute test');
	RETURN;
END_IF

// Setup command with configurations
iTestCommand.InjectConfigurations(
	iComponent := iTestComponent,
	iCommandConfiguration := iTestCommandConfig,
	iPermIntlkConfiguration := iTestPermIntlkConfig
);

// Test 1: Abort command that is currently running (busy)
stBaseStatus.Busy := TRUE;
stBaseStatus.Done := FALSE;
IF iTestCommandConfig <> 0 THEN
	stCommandConfiguration := iTestCommandConfig.P_CommandConfiguration;
END_IF
stCommandStatus.StepState := E_CommandState.Execute;
stCommandStatus.Result := E_CommandResult.Accepted;
iTestCommand.SetCommandStatus(stCommandStatus);

// Verify command is in running state before abort
AssertTrue(
	Condition := iTestCommand.P_CommandStatus.BaseStatus.Busy,
	Message := 'Command should be busy before abort'
);

// Call Abort method
iTestCommand.Abort();

// Verify command was aborted properly
AssertFalse(
	Condition := iTestCommand.P_CommandStatus.BaseStatus.Busy,
	Message := 'Command should not be busy after abort'
);

AssertEquals_UDINT(
	Expected := E_CommandResult.Aborted,
	Actual := iTestCommand.P_CommandStatus.Result,
	Message := 'Command result should be Aborted after calling Abort()'
);

AssertFalse(
	Condition := iTestCommand.P_CommandStatus.BaseStatus.Done,
	Message := 'Command Done flag should be FALSE after abort'
);

// Test 2: Cancel command from Accepted state (queued command)
stBaseStatus.Busy := FALSE;
stBaseStatus.Done := FALSE;
stCommandStatus.BaseStatus REF= stBaseStatus;
IF iTestCommandConfig <> 0 THEN
	stCommandConfiguration := iTestCommandConfig.P_CommandConfiguration;
END_IF
stCommandStatus.StepState := E_CommandState.Idle;
stCommandStatus.Result := E_CommandResult.Accepted;
iTestCommand.SetCommandStatus(stCommandStatus);

iTestCommand.Cancel();

AssertFalse(
	Condition := iTestCommand.P_CommandStatus.BaseStatus.Busy,
	Message := 'Command should not be busy after cancel (from Accepted state)'
);

AssertEquals_UDINT(
	Expected := E_CommandResult.Cancelled,
	Actual := iTestCommand.P_CommandStatus.Result,
	Message := 'Command result should be Cancelled after calling Cancel() from Accepted state'
);

// Test 3: Abort command from Paused state
stBaseStatus.Busy := TRUE;
stBaseStatus.Done := FALSE;
stCommandStatus.BaseStatus REF= stBaseStatus;
IF iTestCommandConfig <> 0 THEN
	stCommandConfiguration := iTestCommandConfig.P_CommandConfiguration;
END_IF
stCommandStatus.StepState := E_CommandState.Paused;
stCommandStatus.Result := E_CommandResult.Accepted;
iTestCommand.SetCommandStatus(stCommandStatus);

iTestCommand.Abort();

AssertEquals_UDINT(
	Expected := E_CommandResult.Aborted,
	Actual := iTestCommand.P_CommandStatus.Result,
	Message := 'Command result should be Aborted after calling Abort() from Paused state'
);

// Test 4: Abort command that is already completed (should preserve terminal result per policy)
stBaseStatus.Busy := FALSE;
stBaseStatus.Done := TRUE;
stCommandStatus.BaseStatus REF= stBaseStatus;
IF iTestCommandConfig <> 0 THEN
	stCommandConfiguration := iTestCommandConfig.P_CommandConfiguration;
END_IF
stCommandStatus.StepState := E_CommandState.Complete;
stCommandStatus.Result := E_CommandResult.OK;
iTestCommand.SetCommandStatus(stCommandStatus);

iTestCommand.Abort();

// Policy: Completed commands preserve their terminal results and cannot be aborted
AssertEquals_UDINT(
	Expected := E_CommandResult.OK,
	Actual := iTestCommand.P_CommandStatus.Result,
	Message := 'Completed command should preserve terminal result when abort is called'
);

AssertTrue(
	Condition := iTestCommand.P_CommandStatus.BaseStatus.Done,
	Message := 'Completed command Done flag should remain TRUE when abort is called'
);

TEST_FINISHED();
END_METHOD

METHOD PRIVATE TEST_Cancel_SetsResultToCancelled
VAR
	TestIdx : DINT := INDEX_CANCEL_SETSRESULTCANCELLED;
	stCommandStatus : ST_CommandStatus;
	stBaseStatus : ST_BaseStatus;
	stCommandConfiguration : ST_CommandConfiguration;
END_VAR
TEST(__POUNAME());
// Purpose: Distinguishes between queued vs. running cancel behavior.
// Impact: Ensures Cancel actually produces the Cancelled result (and not silently ignored).
// Reference: FB_Command.TcPOU Cancel() method and queue management logic

// Initialize reference objects for stCommandStatus
stCommandStatus.BaseStatus REF= stBaseStatus;
stCommandStatus.ConfigRef REF= stCommandConfiguration;

// === TEST SCENARIO 1: Cancel Queued Command ===
// Initialize test objects first - Use index 53 to avoid conflicts
TestCommand[TestIdx].Initialize();
TestComponent[TestIdx].Initialize();
TestCommandConfig[TestIdx].Initialize();
TestPermIntlk[TestIdx].Initialize();

// Safe interface assignments using __QUERYINTERFACE for validation
iTestCommand := TestCommand[TestIdx];

iTestCommandConfig := TestCommandConfig[TestIdx];

iTestComponent := TestComponent[TestIdx];

iTestPermIntlkConfig := TestPermIntlk[TestIdx];

// Configure command for cancel testing
TestCommandConfig[TestIdx].P_CommandConfiguration.CommandDescription := 'Cancel Test - Queued Command';
IF __ISVALIDREF(TestCommandConfig[TestIdx].P_CommandConfiguration.BaseConfiguration) THEN
    TestCommandConfig[TestIdx].P_CommandConfiguration.BaseConfiguration.LogTraceConfiguration.When := E_LogTraceWhen.xRunOnInitOnly;
END_IF

// Configure permissive to be OK for successful validation
IF iTestPermIntlkConfig <> 0 THEN
	iTestPermIntlkConfig.P_PermIntlkConfiguration.PermIntlkObj[1].Description := 'Cancel Test Permissive';
	iTestPermIntlkConfig.P_PermIntlkConfiguration.PermIntlkObj[1].Condition := TRUE;
	iTestPermIntlkConfig.P_PermIntlkConfiguration.PermIntlkObj[1].Index := 1;
END_IF

// Setup command with configurations
iTestCommand.InjectConfigurations(
	iComponent := iTestComponent,
	iCommandConfiguration := iTestCommandConfig,
	iPermIntlkConfiguration := iTestPermIntlkConfig
);

// Queue the command (puts it in queue without executing)
iTestCommand.Queue();

// Verify command is queued
AssertEquals_UDINT(
	Expected := E_CommandState.Idle,
	Actual := iTestCommand.P_CommandStatus.StepState,
	Message := 'QUEUED CANCEL TEST: Queued command should be in Idle state'
);

AssertEquals_UDINT(
	Expected := E_CommandResult.Accepted,
	Actual := iTestCommand.P_CommandStatus.Result,
	Message := 'QUEUED CANCEL TEST: Queued command should have Accepted result'
);

// CRITICAL TEST: Cancel queued command
iTestCommand.Cancel();

// Verify Cancelled result is set for queued command
AssertEquals_UDINT(
	Expected := E_CommandResult.Cancelled,
	Actual := iTestCommand.P_CommandStatus.Result,
	Message := 'QUEUED CANCEL TEST: Cancel() must set Result=Cancelled for queued commands'
);

// Verify command remains in Idle state after cancel
AssertEquals_UDINT(
	Expected := E_CommandState.Idle,
	Actual := iTestCommand.P_CommandStatus.StepState,
	Message := 'QUEUED CANCEL TEST: Cancelled command should remain in Idle state'
);

// Verify flags are set correctly for cancelled queued command
AssertFalse(
	Condition := iTestCommand.P_CommandStatus.BaseStatus.Busy,
	Message := 'QUEUED CANCEL TEST: Cancelled queued command should have Busy=FALSE'
);

